LIN {X 0,Y 254.728,Z 728.451,A -85,B 0,C 180,E1 29641.69,E2 29641.69} C_VEL
LIN {X 0,Y 225.96,Z 695.224,A -85,B 0,C 180,E1 29666.244,E2 29666.244} C_VEL
LIN {X 0,Y 232.999,Z 658.239,A -85,B 0,C 180,E1 29686.941,E2 29686.941} C_VEL
LIN {X 0,Y 236.204,Z 647.926,A -85,B 0,C 180,E1 29697.112,E2 29697.112} C_VEL
LIN {X 0,Y 235.985,Z 649.701,A -85,B 0,C 180,E1 29705.085,E2 29705.085} C_VEL
LIN {X 0,Y 233.22,Z 662.932,A -85,B 0,C 180,E1 29715.199,E2 29715.199} C_VEL
LIN {X 0,Y 229.881,Z 671.076,A -85,B 0,C 180,E1 29718.505,E2 29718.505} C_VEL
LIN {X 0,Y 187.85,Z 714.712,A -85,B 0,C 180,E1 29726.634,E2 29726.634} C_VEL
LIN {X 0,Y 147.086,Z 745.833,A -85,B 0,C 180,E1 29741.377,E2 29741.377} C_VEL
LIN {X 0,Y 119.441,Z 763.935,A -85,B 0,C 180,E1 29767.61,E2 29767.61} C_VEL
LIN {X 0,Y 115.488,Z 767.444,A -85,B 0,C 180,E1 29793.764,E2 29793.764} C_VEL
LIN {X 0,Y 126.212,Z 759.493,A -85,B 0,C 180,E1 29822.73,E2 29822.73} C_VEL
LIN {X 0,Y 159.049,Z 737.597,A -85,B 0,C 180,E1 29844.139,E2 29844.139} C_VEL
LIN {X 0,Y 202.331,Z 701.352,A -85,B 0,C 180,E1 29856.657,E2 29856.657} C_VEL
LIN {X 0,Y 232.022,Z 667.67,A -85,B 0,C 180,E1 29862.272,E2 29862.272} C_VEL
LIN {X 0,Y 235.351,Z 652.826,A -85,B 0,C 180,E1 29871.562,E2 29871.562} C_VEL
LIN {X 0,Y 236.575,Z 647.685,A -85,B 0,C 180,E1 29878.052,E2 29878.052} C_VEL
LIN {X 0,Y 235.139,Z 650.478,A -85,B 0,C 180,E1 29886.517,E2 29886.517} C_VEL
LIN {X 0,Y 230.962,Z 664.925,A -85,B 0,C 180,E1 29897.076,E2 29897.076} C_VEL
LIN {X 0,Y 228.751,Z 702.6,A -85,B 0,C 180,E1 29918.911,E2 29918.911} C_VEL
LIN {X 0,Y 256.269,Z 729.185,A -85,B 0,C 180,E1 29938.946,E2 29938.946} C_VEL
LIN {X 0,Y 277.902,Z 744.199,A -85,B 0,C 180,E1 29950.33,E2 29950.33} C_VEL
LIN {X 0,Y 291.233,Z 754.024,A -85,B 0,C 180,E1 29959.499,E2 29959.499} C_VEL
LIN {X 0,Y 297.321,Z 758.46,A -85,B 0,C 180,E1 29968.539,E2 29968.539} C_VEL
LIN {X 0,Y 293.962,Z 756.258,A -85,B 0,C 180,E1 29977.41,E2 29977.41} C_VEL
LIN {X 0,Y 285.173,Z 749.557,A -85,B 0,C 180,E1 29985.141,E2 29985.141} C_VEL
LIN {X 0,Y 267.259,Z 737.135,A -85,B 0,C 180,E1 29995.187,E2 29995.187} C_VEL
LIN {X 0,Y 254.728,Z 728.451,A -85,B 0,C 180,E1 30001.69,E2 30001.69} C_VEL
LIN {X 0,Y 235.39,Z 722.248,A -85,B 0,C 180,E1 30008.545,E2 30008.545} C_VEL
LIN {X 0,Y 219.271,Z 687.766,A -85,B 0,C 180,E1 30034.122,E2 30034.122} C_VEL
LIN {X 0,Y 227.812,Z 663.177,A -85,B 0,C 180,E1 30047.874,E2 30047.874} C_VEL
LIN {X 0,Y 231.564,Z 653.613,A -85,B 0,C 180,E1 30058.235,E2 30058.235} C_VEL
LIN {X 0,Y 230.318,Z 658.459,A -85,B 0,C 180,E1 30067.685,E2 30067.685} C_VEL
LIN {X 0,Y 226.212,Z 672.442,A -85,B 0,C 180,E1 30076.746,E2 30076.746} C_VEL
LIN {X 0,Y 182.571,Z 716.057,A -85,B 0,C 180,E1 30084.791,E2 30084.791} C_VEL
LIN {X 0,Y 139.135,Z 747.341,A -85,B 0,C 180,E1 30100.274,E2 30100.274} C_VEL
LIN {X 0,Y 111.968,Z 763.757,A -85,B 0,C 180,E1 30126.026,E2 30126.026} C_VEL
LIN {X 0,Y 107.486,Z 767.269,A -85,B 0,C 180,E1 30154.045,E2 30154.045} C_VEL
LIN {X 0,Y 119.424,Z 759.314,A -85,B 0,C 180,E1 30184.849,E2 30184.849} C_VEL
LIN {X 0,Y 156.677,Z 735.903,A -85,B 0,C 180,E1 30207.488,E2 30207.488} C_VEL
LIN {X 0,Y 202.506,Z 698.173,A -85,B 0,C 180,E1 30219.402,E2 30219.402} C_VEL
LIN {X 0,Y 226.779,Z 671.402,A -85,B 0,C 180,E1 30223.58,E2 30223.58} C_VEL
LIN {X 0,Y 230.339,Z 658.433,A -85,B 0,C 180,E1 30232.316,E2 30232.316} C_VEL
LIN {X 0,Y 231.466,Z 653.736,A -85,B 0,C 180,E1 30241.766,E2 30241.766} C_VEL
LIN {X 0,Y 227.823,Z 663.166,A -85,B 0,C 180,E1 30252.127,E2 30252.127} C_VEL
LIN {X 0,Y 221.662,Z 706.254,A -85,B 0,C 180,E1 30278.627,E2 30278.627} C_VEL
LIN {X 0,Y 249.251,Z 732.077,A -85,B 0,C 180,E1 30299.507,E2 30299.507} C_VEL
LIN {X 0,Y 270.249,Z 745.742,A -85,B 0,C 180,E1 30310.718,E2 30310.718} C_VEL
LIN {X 0,Y 284.074,Z 755.281,A -85,B 0,C 180,E1 30320.563,E2 30320.563} C_VEL
LIN {X 0,Y 289.26,Z 758.636,A -85,B 0,C 180,E1 30328.498,E2 30328.498} C_VEL
LIN {X 0,Y 287.734,Z 757.916,A -85,B 0,C 180,E1 30334.534,E2 30334.534} C_VEL
LIN {X 0,Y 281.099,Z 753.131,A -85,B 0,C 180,E1 30342.16,E2 30342.16} C_VEL
LIN {X 0,Y 265.437,Z 742.878,A -85,B 0,C 180,E1 30351.799,E2 30351.799} C_VEL
LIN {X 0,Y 239.784,Z 725.609,A -85,B 0,C 180,E1 30365.759,E2 30365.759} C_VEL
LIN {X 0,Y 235.39,Z 722.248,A -85,B 0,C 180,E1 30368.545,E2 30368.545} C_VEL
LIN {X 0,Y 218.325,Z 716.283,A -85,B 0,C 180,E1 30376.29,E2 30376.29} C_VEL
LIN {X 0,Y 216.594,Z 681.525,A -85,B 0,C 180,E1 30400.946,E2 30400.946} C_VEL
LIN {X 0,Y 223.467,Z 666.107,A -85,B 0,C 180,E1 30410.346,E2 30410.346} C_VEL
LIN {X 0,Y 226.478,Z 659.971,A -85,B 0,C 180,E1 30418.196,E2 30418.196} C_VEL
LIN {X 0,Y 225.418,Z 663.045,A -85,B 0,C 180,E1 30425.911,E2 30425.911} C_VEL
LIN {X 0,Y 221.713,Z 674.444,A -85,B 0,C 180,E1 30434.56,E2 30434.56} C_VEL
LIN {X 0,Y 178.102,Z 716.889,A -85,B 0,C 180,E1 30442.7,E2 30442.7} C_VEL
LIN {X 0,Y 134.023,Z 747.163,A -85,B 0,C 180,E1 30457.621,E2 30457.621} C_VEL
LIN {X 0,Y 104.613,Z 763.58,A -85,B 0,C 180,E1 30484.222,E2 30484.222} C_VEL
LIN {X 0,Y 99.454,Z 767.059,A -85,B 0,C 180,E1 30515.015,E2 30515.015} C_VEL
LIN {X 0,Y 114.521,Z 758.116,A -85,B 0,C 180,E1 30548.976,E2 30548.976} C_VEL
LIN {X 0,Y 153.452,Z 735.034,A -85,B 0,C 180,E1 30570.429,E2 30570.429} C_VEL
LIN {X 0,Y 199.79,Z 697.995,A -85,B 0,C 180,E1 30581.586,E2 30581.586} C_VEL
LIN {X 0,Y 221.953,Z 674.175,A -85,B 0,C 180,E1 30585.469,E2 30585.469} C_VEL
LIN {X 0,Y 225.412,Z 663.051,A -85,B 0,C 180,E1 30594.089,E2 30594.089} C_VEL
LIN {X 0,Y 226.375,Z 660.091,A -85,B 0,C 180,E1 30601.805,E2 30601.805} C_VEL
LIN {X 0,Y 221.763,Z 670.312,A -85,B 0,C 180,E1 30612.726,E2 30612.726} C_VEL
LIN {X 0,Y 214.375,Z 709.528,A -85,B 0,C 180,E1 30638.119,E2 30638.119} C_VEL
LIN {X 0,Y 242.903,Z 735.294,A -85,B 0,C 180,E1 30660.516,E2 30660.516} C_VEL
LIN {X 0,Y 263.361,Z 747.739,A -85,B 0,C 180,E1 30671.592,E2 30671.592} C_VEL
LIN {X 0,Y 275.604,Z 755.471,A -85,B 0,C 180,E1 30680.271,E2 30680.271} C_VEL
LIN {X 0,Y 281.172,Z 758.813,A -85,B 0,C 180,E1 30688.455,E2 30688.455} C_VEL
LIN {X 0,Y 279.558,Z 758.096,A -85,B 0,C 180,E1 30694.667,E2 30694.667} C_VEL
LIN {X 0,Y 271.859,Z 753.075,A -85,B 0,C 180,E1 30702.843,E2 30702.843} C_VEL
LIN {X 0,Y 254.88,Z 742.852,A -85,B 0,C 180,E1 30712.945,E2 30712.945} C_VEL
LIN {X 0,Y 227.506,Z 724.851,A -85,B 0,C 180,E1 30728.684,E2 30728.684} C_VEL
LIN {X 0,Y 218.325,Z 716.283,A -85,B 0,C 180,E1 30736.29,E2 30736.29} C_VEL
LIN {X 0,Y 205.918,Z 709.678,A -85,B 0,C 180,E1 30745.1,E2 30745.1} C_VEL
LIN {X 0,Y 217.606,Z 672.647,A -85,B 0,C 180,E1 30770.083,E2 30770.083} C_VEL
LIN {X 0,Y 221.058,Z 666.041,A -85,B 0,C 180,E1 30778.151,E2 30778.151} C_VEL
LIN {X 0,Y 219.856,Z 669.284,A -85,B 0,C 180,E1 30786.061,E2 30786.061} C_VEL
LIN {X 0,Y 216.387,Z 678.218,A -85,B 0,C 180,E1 30793.213,E2 30793.213} C_VEL
LIN {X 0,Y 170.784,Z 720.013,A -85,B 0,C 180,E1 30801.194,E2 30801.194} C_VEL
LIN {X 0,Y 124.008,Z 749.858,A -85,B 0,C 180,E1 30817.356,E2 30817.356} C_VEL
LIN {X 0,Y 95.225,Z 764.536,A -85,B 0,C 180,E1 30846.538,E2 30846.538} C_VEL
LIN {X 0,Y 91.484,Z 766.918,A -85,B 0,C 180,E1 30874.754,E2 30874.754} C_VEL
LIN {X 0,Y 106.426,Z 758.957,A -85,B 0,C 180,E1 30909.882,E2 30909.882} C_VEL
LIN {X 0,Y 148.984,Z 735.263,A -85,B 0,C 180,E1 30932.955,E2 30932.955} C_VEL
LIN {X 0,Y 197.378,Z 697.818,A -85,B 0,C 180,E1 30943.821,E2 30943.821} C_VEL
LIN {X 0,Y 216.834,Z 677.517,A -85,B 0,C 180,E1 30947.079,E2 30947.079} C_VEL
LIN {X 0,Y 220.44,Z 667.708,A -85,B 0,C 180,E1 30955.951,E2 30955.951} C_VEL
LIN {X 0,Y 220.308,Z 667.079,A -85,B 0,C 180,E1 30963.529,E2 30963.529} C_VEL
LIN {X 0,Y 215.403,Z 676.961,A -85,B 0,C 180,E1 30973.109,E2 30973.109} C_VEL
LIN {X 0,Y 207.451,Z 713.563,A -85,B 0,C 180,E1 30998.277,E2 30998.277} C_VEL
LIN {X 0,Y 235.856,Z 737.914,A -85,B 0,C 180,E1 31021.169,E2 31021.169} C_VEL
LIN {X 0,Y 256.839,Z 749.754,A -85,B 0,C 180,E1 31032.751,E2 31032.751} C_VEL
LIN {X 0,Y 268.905,Z 756.817,A -85,B 0,C 180,E1 31041.895,E2 31041.895} C_VEL
LIN {X 0,Y 273.109,Z 758.99,A -85,B 0,C 180,E1 31048.409,E2 31048.409} C_VEL
LIN {X 0,Y 271.34,Z 758.278,A -85,B 0,C 180,E1 31054.809,E2 31054.809} C_VEL
LIN {X 0,Y 262.883,Z 753.278,A -85,B 0,C 180,E1 31063.289,E2 31063.289} C_VEL
LIN {X 0,Y 245.026,Z 743.359,A -85,B 0,C 180,E1 31073.722,E2 31073.722} C_VEL
LIN {X 0,Y 217.8,Z 726.02,A -85,B 0,C 180,E1 31090.169,E2 31090.169} C_VEL
LIN {X 0,Y 205.918,Z 709.678,A -85,B 0,C 180,E1 31105.1,E2 31105.1} C_VEL
LIN {X 0,Y 199.485,Z 701.993,A -85,B 0,C 180,E1 31114.737,E2 31114.737} C_VEL
LIN {X 0,Y 212.093,Z 677.669,A -85,B 0,C 180,E1 31130.862,E2 31130.862} C_VEL
LIN {X 0,Y 215.64,Z 672.089,A -85,B 0,C 180,E1 31138.105,E2 31138.105} C_VEL
LIN {X 0,Y 214.136,Z 675.443,A -85,B 0,C 180,E1 31146.223,E2 31146.223} C_VEL
LIN {X 0,Y 210.393,Z 682.827,A -85,B 0,C 180,E1 31151.881,E2 31151.881} C_VEL
LIN {X 0,Y 163.045,Z 723.354,A -85,B 0,C 180,E1 31159.655,E2 31159.655} C_VEL
LIN {X 0,Y 116.019,Z 751.214,A -85,B 0,C 180,E1 31175.896,E2 31175.896} C_VEL
LIN {X 0,Y 87.861,Z 764.36,A -85,B 0,C 180,E1 31204.437,E2 31204.437} C_VEL
LIN {X 0,Y 83.47,Z 766.742,A -85,B 0,C 180,E1 31235.211,E2 31235.211} C_VEL
LIN {X 0,Y 100.289,Z 758.779,A -85,B 0,C 180,E1 31272.879,E2 31272.879} C_VEL
LIN {X 0,Y 145.43,Z 735.084,A -85,B 0,C 180,E1 31295.841,E2 31295.841} C_VEL
LIN {X 0,Y 195.273,Z 697.641,A -85,B 0,C 180,E1 31306.106,E2 31306.106} C_VEL
LIN {X 0,Y 211.826,Z 680.845,A -85,B 0,C 180,E1 31308.851,E2 31308.851} C_VEL
LIN {X 0,Y 215.556,Z 672.545,A -85,B 0,C 180,E1 31317.862,E2 31317.862} C_VEL
LIN {X 0,Y 213.738,Z 674.762,A -85,B 0,C 180,E1 31325.99,E2 31325.99} C_VEL
LIN {X 0,Y 206.613,Z 687.133,A -85,B 0,C 180,E1 31335.63,E2 31335.63} C_VEL
LIN {X 0,Y 201.148,Z 718.649,A -85,B 0,C 180,E1 31359.708,E2 31359.708} C_VEL
LIN {X 0,Y 230.107,Z 741.108,A -85,B 0,C 180,E1 31382.642,E2 31382.642} C_VEL
LIN {X 0,Y 250.759,Z 751.859,A -85,B 0,C 180,E1 31394.208,E2 31394.208} C_VEL
LIN {X 0,Y 260.559,Z 757.003,A -85,B 0,C 180,E1 31401.634,E2 31401.634} C_VEL
LIN {X 0,Y 265.004,Z 759.167,A -85,B 0,C 180,E1 31408.361,E2 31408.361} C_VEL
LIN {X 0,Y 263.113,Z 758.46,A -85,B 0,C 180,E1 31414.96,E2 31414.96} C_VEL
LIN {X 0,Y 253.467,Z 753.325,A -85,B 0,C 180,E1 31423.971,E2 31423.971} C_VEL
LIN {X 0,Y 234.404,Z 743.612,A -85,B 0,C 180,E1 31434.868,E2 31434.868} C_VEL
LIN {X 0,Y 205.25,Z 724.518,A -85,B 0,C 180,E1 31454.581,E2 31454.581} C_VEL
LIN {X 0,Y 199.485,Z 701.993,A -85,B 0,C 180,E1 31474.737,E2 31474.737} C_VEL
LIN {X 0,Y 199.798,Z 692.818,A -85,B 0,C 180,E1 31484.582,E2 31484.582} C_VEL
LIN {X 0,Y 207.901,Z 680.595,A -85,B 0,C 180,E1 31493.841,E2 31493.841} C_VEL
LIN {X 0,Y 209.887,Z 677.873,A -85,B 0,C 180,E1 31498.053,E2 31498.053} C_VEL
LIN {X 0,Y 208.209,Z 681.369,A -85,B 0,C 180,E1 31506.401,E2 31506.401} C_VEL
LIN {X 0,Y 204.322,Z 687.264,A -85,B 0,C 180,E1 31510.23,E2 31510.23} C_VEL
LIN {X 0,Y 155.19,Z 726.857,A -85,B 0,C 180,E1 31518.046,E2 31518.046} C_VEL
LIN {X 0,Y 106.489,Z 753.364,A -85,B 0,C 180,E1 31535.189,E2 31535.189} C_VEL
LIN {X 0,Y 76.779,Z 765.765,A -85,B 0,C 180,E1 31572.766,E2 31572.766} C_VEL
LIN {X 0,Y 76.798,Z 765.765,A -85,B 0,C 180,E1 31607.229,E2 31607.229} C_VEL
LIN {X 0,Y 106.401,Z 753.393,A -85,B 0,C 180,E1 31644.793,E2 31644.793} C_VEL
LIN {X 0,Y 156.662,Z 725.837,A -85,B 0,C 180,E1 31662.297,E2 31662.297} C_VEL
LIN {X 0,Y 206.169,Z 685.486,A -85,B 0,C 180,E1 31670,E2 31670} C_VEL
LIN {X 0,Y 209.786,Z 678.334,A -85,B 0,C 180,E1 31677.803,E2 31677.803} C_VEL
LIN {X 0,Y 208.766,Z 679.221,A -85,B 0,C 180,E1 31684.043,E2 31684.043} C_VEL
LIN {X 0,Y 202.748,Z 688.544,A -85,B 0,C 180,E1 31692.9,E2 31692.9} C_VEL
LIN {X 0,Y 193.386,Z 721.096,A -85,B 0,C 180,E1 31718.661,E2 31718.661} C_VEL
LIN {X 0,Y 220.27,Z 741.933,A -85,B 0,C 180,E1 31741.778,E2 31741.778} C_VEL
LIN {X 0,Y 243.246,Z 752.979,A -85,B 0,C 180,E1 31754.78,E2 31754.78} C_VEL
LIN {X 0,Y 252.476,Z 757.404,A -85,B 0,C 180,E1 31761.786,E2 31761.786} C_VEL
LIN {X 0,Y 256.875,Z 759.345,A -85,B 0,C 180,E1 31768.309,E2 31768.309} C_VEL
LIN {X 0,Y 254.845,Z 758.642,A -85,B 0,C 180,E1 31775.121,E2 31775.121} C_VEL
LIN {X 0,Y 245.339,Z 754.088,A -85,B 0,C 180,E1 31783.771,E2 31783.771} C_VEL
LIN {X 0,Y 225.561,Z 744.821,A -85,B 0,C 180,E1 31795.035,E2 31795.035} C_VEL
LIN {X 0,Y 196.549,Z 726.274,A -85,B 0,C 180,E1 31815.926,E2 31815.926} C_VEL
LIN {X 0,Y 198.212,Z 695.345,A -85,B 0,C 180,E1 31843.011,E2 31843.011} C_VEL
LIN {X 0,Y 199.798,Z 692.818,A -85,B 0,C 180,E1 31844.582,E2 31844.582} C_VEL
LIN {X 0,Y 202.236,Z 685.819,A -85,B 0,C 180,E1 31854.611,E2 31854.611} C_VEL
LIN {X 0,Y 204.067,Z 683.66,A -85,B 0,C 180,E1 31857.997,E2 31857.997} C_VEL
LIN {X 0,Y 203.221,Z 685.374,A -85,B 0,C 180,E1 31864.215,E2 31864.215} C_VEL
LIN {X 0,Y 199.657,Z 690.226,A -85,B 0,C 180,E1 31868.341,E2 31868.341} C_VEL
LIN {X 0,Y 147.973,Z 729.601,A -85,B 0,C 180,E1 31876.098,E2 31876.098} C_VEL
LIN {X 0,Y 96.642,Z 755.344,A -85,B 0,C 180,E1 31894.53,E2 31894.53} C_VEL
LIN {X 0,Y 69.101,Z 765.588,A -85,B 0,C 180,E1 31930.78,E2 31930.78} C_VEL
LIN {X 0,Y 69.137,Z 765.589,A -85,B 0,C 180,E1 31969.209,E2 31969.209} C_VEL
LIN {X 0,Y 102.069,Z 753.138,A -85,B 0,C 180,E1 32008.647,E2 32008.647} C_VEL
LIN {X 0,Y 154.28,Z 725.724,A -85,B 0,C 180,E1 32025.167,E2 32025.167} C_VEL
LIN {X 0,Y 201.651,Z 688.062,A -85,B 0,C 180,E1 32032.501,E2 32032.501} C_VEL
LIN {X 0,Y 203.979,Z 684.108,A -85,B 0,C 180,E1 32037.741,E2 32037.741} C_VEL
LIN {X 0,Y 203.077,Z 684.785,A -85,B 0,C 180,E1 32043.757,E2 32043.757} C_VEL
LIN {X 0,Y 196.291,Z 693.939,A -85,B 0,C 180,E1 32052.561,E2 32052.561} C_VEL
LIN {X 0,Y 186.512,Z 725.125,A -85,B 0,C 180,E1 32079.428,E2 32079.428} C_VEL
LIN {X 0,Y 216.109,Z 745.558,A -85,B 0,C 180,E1 32104.259,E2 32104.259} C_VEL
LIN {X 0,Y 234.036,Z 753.325,A -85,B 0,C 180,E1 32114.324,E2 32114.324} C_VEL
LIN {X 0,Y 243.304,Z 757.389,A -85,B 0,C 180,E1 32121.036,E2 32121.036} C_VEL
LIN {X 0,Y 248.744,Z 759.522,A -85,B 0,C 180,E1 32128.253,E2 32128.253} C_VEL
LIN {X 0,Y 246.557,Z 758.825,A -85,B 0,C 180,E1 32135.294,E2 32135.294} C_VEL
LIN {X 0,Y 238.261,Z 755.22,A -85,B 0,C 180,E1 32142.872,E2 32142.872} C_VEL
LIN {X 0,Y 218.727,Z 746.935,A -85,B 0,C 180,E1 32154.094,E2 32154.094} C_VEL
LIN {X 0,Y 189.194,Z 729.369,A -85,B 0,C 180,E1 32175.802,E2 32175.802} C_VEL
LIN {X 0,Y 192.268,Z 699.14,A -85,B 0,C 180,E1 32204.108,E2 32204.108} C_VEL
LIN {X 0,Y 201.715,Z 686.519,A -85,B 0,C 180,E1 32213.652,E2 32213.652} C_VEL
LIN {X 0,Y 202.236,Z 685.819,A -85,B 0,C 180,E1 32214.611,E2 32214.611} C_VEL
LIN {X 0,Y 199.741,Z 687.736,A -85,B 0,C 180,E1 32220.845,E2 32220.845} C_VEL
LIN {X 0,Y 196.779,Z 691.204,A -85,B 0,C 180,E1 32224.687,E2 32224.687} C_VEL
LIN {X 0,Y 192.694,Z 695.503,A -85,B 0,C 180,E1 32226.61,E2 32226.61} C_VEL
LIN {X 0,Y 140.689,Z 732.503,A -85,B 0,C 180,E1 32234.042,E2 32234.042} C_VEL
LIN {X 0,Y 89.421,Z 756.194,A -85,B 0,C 180,E1 32252.01,E2 32252.01} C_VEL
LIN {X 0,Y 61.525,Z 765.411,A -85,B 0,C 180,E1 32288.301,E2 32288.301} C_VEL
LIN {X 0,Y 61.555,Z 765.412,A -85,B 0,C 180,E1 32331.687,E2 32331.687} C_VEL
LIN {X 0,Y 98.096,Z 752.949,A -85,B 0,C 180,E1 32372.735,E2 32372.735} C_VEL
LIN {X 0,Y 151.716,Z 725.995,A -85,B 0,C 180,E1 32388.019,E2 32388.019} C_VEL
LIN {X 0,Y 196.221,Z 692.141,A -85,B 0,C 180,E1 32394.061,E2 32394.061} C_VEL
LIN {X 0,Y 197.827,Z 689.304,A -85,B 0,C 180,E1 32402.066,E2 32402.066} C_VEL
LIN {X 0,Y 190.666,Z 697.871,A -85,B 0,C 180,E1 32411.335,E2 32411.335} C_VEL
LIN {X 0,Y 179.083,Z 728.149,A -85,B 0,C 180,E1 32439.262,E2 32439.262} C_VEL
LIN {X 0,Y 208.813,Z 747.467,A -85,B 0,C 180,E1 32464.966,E2 32464.966} C_VEL
LIN {X 0,Y 228.932,Z 755.432,A -85,B 0,C 180,E1 32476.594,E2 32476.594} C_VEL
LIN {X 0,Y 238.105,Z 759.012,A -85,B 0,C 180,E1 32484.518,E2 32484.518} C_VEL
LIN {X 0,Y 240.556,Z 759.702,A -85,B 0,C 180,E1 32491.806,E2 32491.806} C_VEL
LIN {X 0,Y 232.853,Z 756.938,A -85,B 0,C 180,E1 32500.695,E2 32500.695} C_VEL
LIN {X 0,Y 214.366,Z 749.866,A -85,B 0,C 180,E1 32511.754,E2 32511.754} C_VEL
LIN {X 0,Y 184.349,Z 734.606,A -85,B 0,C 180,E1 32532.559,E2 32532.559} C_VEL
LIN {X 0,Y 184.485,Z 705.482,A -85,B 0,C 180,E1 32563.419,E2 32563.419} C_VEL
LIN {X 0,Y 195.211,Z 692.31,A -85,B 0,C 180,E1 32573.439,E2 32573.439} C_VEL
LIN {X 0,Y 197.972,Z 689.176,A -85,B 0,C 180,E1 32577.936,E2 32577.936} C_VEL
LIN {X 0,Y 196.779,Z 691.204,A -85,B 0,C 180,E1 32584.687,E2 32584.687} C_VEL
LIN {X 0,Y 189.449,Z 697.862,A -85,B 0,C 180,E1 32585.726,E2 32585.726} C_VEL
LIN {X 0,Y 178.401,Z 706.412,A -85,B 0,C 180,E1 32585.494,E2 32585.494} C_VEL
LIN {X 0,Y 124.402,Z 739.949,A -85,B 0,C 180,E1 32593.744,E2 32593.744} C_VEL
LIN {X 0,Y 74.046,Z 759.677,A -85,B 0,C 180,E1 32614.993,E2 32614.993} C_VEL
LIN {X 0,Y 51.354,Z 766.036,A -85,B 0,C 180,E1 32661.508,E2 32661.508} C_VEL
LIN {X 0,Y 64.306,Z 762.508,A -85,B 0,C 180,E1 32715.079,E2 32715.079} C_VEL
LIN {X 0,Y 114.509,Z 744.576,A -85,B 0,C 180,E1 32743.768,E2 32743.768} C_VEL
LIN {X 0,Y 169.769,Z 712.734,A -85,B 0,C 180,E1 32753.594,E2 32753.594} C_VEL
LIN {X 0,Y 190.108,Z 696.931,A -85,B 0,C 180,E1 32755.649,E2 32755.649} C_VEL
LIN {X 0,Y 191.615,Z 694.804,A -85,B 0,C 180,E1 32762.133,E2 32762.133} C_VEL
LIN {X 0,Y 183.803,Z 703.06,A -85,B 0,C 180,E1 32771.024,E2 32771.024} C_VEL
LIN {X 0,Y 171.752,Z 731.326,A -85,B 0,C 180,E1 32799.352,E2 32799.352} C_VEL
LIN {X 0,Y 201.111,Z 749.136,A -85,B 0,C 180,E1 32825.498,E2 32825.498} C_VEL
LIN {X 0,Y 219.601,Z 755.644,A -85,B 0,C 180,E1 32836.013,E2 32836.013} C_VEL
LIN {X 0,Y 229.721,Z 759.198,A -85,B 0,C 180,E1 32844.317,E2 32844.317} C_VEL
LIN {X 0,Y 232.372,Z 759.881,A -85,B 0,C 180,E1 32851.87,E2 32851.87} C_VEL
LIN {X 0,Y 223.718,Z 757.164,A -85,B 0,C 180,E1 32861.089,E2 32861.089} C_VEL
LIN {X 0,Y 204.565,Z 750.536,A -85,B 0,C 180,E1 32872.351,E2 32872.351} C_VEL
LIN {X 0,Y 173.957,Z 734.75,A -85,B 0,C 180,E1 32895.966,E2 32895.966} C_VEL
LIN {X 0,Y 180.883,Z 706.241,A -85,B 0,C 180,E1 32926.825,E2 32926.825} C_VEL
LIN {X 0,Y 190.185,Z 696.278,A -85,B 0,C 180,E1 32935.36,E2 32935.36} C_VEL
LIN {X 0,Y 191.692,Z 695.097,A -85,B 0,C 180,E1 32942.404,E2 32942.404} C_VEL
LIN {X 0,Y 188.731,Z 698.051,A -85,B 0,C 180,E1 32944.498,E2 32944.498} C_VEL
LIN {X 0,Y 178.401,Z 706.412,A -85,B 0,C 180,E1 32945.494,E2 32945.494} C_VEL
LIN {X 0,Y 148.742,Z 725.885,A -85,B 0,C 180,E1 32945.933,E2 32945.933} C_VEL
LIN {X 0,Y 91.802,Z 752.594,A -85,B 0,C 180,E1 32958.221,E2 32958.221} C_VEL
LIN {X 0,Y 46.888,Z 765.058,A -85,B 0,C 180,E1 33000.977,E2 33000.977} C_VEL
LIN {X 0,Y 43.565,Z 765.863,A -85,B 0,C 180,E1 33040.022,E2 33040.022} C_VEL
LIN {X 0,Y 75.652,Z 757.886,A -85,B 0,C 180,E1 33094.428,E2 33094.428} C_VEL
LIN {X 0,Y 134.004,Z 734.192,A -85,B 0,C 180,E1 33111.976,E2 33111.976} C_VEL
LIN {X 0,Y 185.409,Z 700.088,A -85,B 0,C 180,E1 33118.165,E2 33118.165} C_VEL
LIN {X 0,Y 183.373,Z 701.639,A -85,B 0,C 180,E1 33124.642,E2 33124.642} C_VEL
LIN {X 0,Y 164.671,Z 734.777,A -85,B 0,C 180,E1 33160.254,E2 33160.254} C_VEL
LIN {X 0,Y 191.794,Z 750.093,A -85,B 0,C 180,E1 33185.142,E2 33185.142} C_VEL
LIN {X 0,Y 210.67,Z 756.171,A -85,B 0,C 180,E1 33195.952,E2 33195.952} C_VEL
LIN {X 0,Y 221.161,Z 759.387,A -85,B 0,C 180,E1 33204.097,E2 33204.097} C_VEL
LIN {X 0,Y 224.192,Z 760.059,A -85,B 0,C 180,E1 33208.062,E2 33208.062} C_VEL
LIN {X 0,Y 221.233,Z 759.385,A -85,B 0,C 180,E1 33215.902,E2 33215.902} C_VEL
LIN {X 0,Y 209.356,Z 755.878,A -85,B 0,C 180,E1 33224.686,E2 33224.686} C_VEL
LIN {X 0,Y 183.378,Z 747.07,A -85,B 0,C 180,E1 33239.973,E2 33239.973} C_VEL
LIN {X 0,Y 164.632,Z 722.855,A -85,B 0,C 180,E1 33275.673,E2 33275.673} C_VEL
LIN {X 0,Y 183.343,Z 701.686,A -85,B 0,C 180,E1 33295.187,E2 33295.187} C_VEL
LIN {X 0,Y 185.414,Z 700.057,A -85,B 0,C 180,E1 33301.654,E2 33301.654} C_VEL
LIN {X 0,Y 148.742,Z 725.885,A -85,B 0,C 180,E1 33305.933,E2 33305.933} C_VEL
LIN {X 0,Y 117.077,Z 741.688,A -85,B 0,C 180,E1 33307,E2 33307} C_VEL
LIN {X 0,Y 59.86,Z 760.913,A -85,B 0,C 180,E1 33327.539,E2 33327.539} C_VEL
LIN {X 0,Y 35.511,Z 765.684,A -85,B 0,C 180,E1 33377.67,E2 33377.67} C_VEL
LIN {X 0,Y 54.025,Z 762.158,A -85,B 0,C 180,E1 33447.362,E2 33447.362} C_VEL
LIN {X 0,Y 110.58,Z 744.422,A -85,B 0,C 180,E1 33471.769,E2 33471.769} C_VEL
LIN {X 0,Y 168.73,Z 712.378,A -85,B 0,C 180,E1 33479.096,E2 33479.096} C_VEL
LIN {X 0,Y 178.953,Z 704.942,A -85,B 0,C 180,E1 33480.308,E2 33480.308} C_VEL
LIN {X 0,Y 172.555,Z 710.349,A -85,B 0,C 180,E1 33488.221,E2 33488.221} C_VEL
LIN {X 0,Y 156.632,Z 736.634,A -85,B 0,C 180,E1 33518.809,E2 33518.809} C_VEL
LIN {X 0,Y 187.745,Z 752.829,A -85,B 0,C 180,E1 33547.96,E2 33547.96} C_VEL
LIN {X 0,Y 207.682,Z 758.303,A -85,B 0,C 180,E1 33559.753,E2 33559.753} C_VEL
LIN {X 0,Y 215.919,Z 760.24,A -85,B 0,C 180,E1 33567.988,E2 33567.988} C_VEL
LIN {X 0,Y 215.903,Z 760.241,A -85,B 0,C 180,E1 33572.013,E2 33572.013} C_VEL
LIN {X 0,Y 207.161,Z 758.199,A -85,B 0,C 180,E1 33580.545,E2 33580.545} C_VEL
LIN {X 0,Y 187.604,Z 752.925,A -85,B 0,C 180,E1 33591.934,E2 33591.934} C_VEL
LIN {X 0,Y 155.715,Z 735.029,A -85,B 0,C 180,E1 33623.894,E2 33623.894} C_VEL
LIN {X 0,Y 176.85,Z 706.721,A -85,B 0,C 180,E1 33655.427,E2 33655.427} C_VEL
LIN {X 0,Y 178.981,Z 704.92,A -85,B 0,C 180,E1 33659.705,E2 33659.705} C_VEL
LIN {X 0,Y 122.023,Z 739.366,A -85,B 0,C 180,E1 33666.153,E2 33666.153} C_VEL
LIN {X 0,Y 117.077,Z 741.688,A -85,B 0,C 180,E1 33667,E2 33667} C_VEL
LIN {X 0,Y 83.788,Z 753.608,A -85,B 0,C 180,E1 33669.138,E2 33669.138} C_VEL
LIN {X 0,Y 33.685,Z 764.705,A -85,B 0,C 180,E1 33707.522,E2 33707.522} C_VEL
LIN {X 0,Y 27.834,Z 765.511,A -85,B 0,C 180,E1 33765.807,E2 33765.807} C_VEL
LIN {X 0,Y 70.172,Z 757.53,A -85,B 0,C 180,E1 33826.529,E2 33826.529} C_VEL
LIN {X 0,Y 132.353,Z 734.018,A -85,B 0,C 180,E1 33838.925,E2 33838.925} C_VEL
LIN {X 0,Y 171.576,Z 710.274,A -85,B 0,C 180,E1 33842.382,E2 33842.382} C_VEL
LIN {X 0,Y 149.878,Z 740.457,A -85,B 0,C 180,E1 33880.917,E2 33880.917} C_VEL
LIN {X 0,Y 177.92,Z 753.555,A -85,B 0,C 180,E1 33907.446,E2 33907.446} C_VEL
LIN {X 0,Y 197.822,Z 758.409,A -85,B 0,C 180,E1 33918.951,E2 33918.951} C_VEL
LIN {X 0,Y 207.589,Z 760.422,A -85,B 0,C 180,E1 33927.907,E2 33927.907} C_VEL
LIN {X 0,Y 205.187,Z 760.058,A -85,B 0,C 180,E1 33935.118,E2 33935.118} C_VEL
LIN {X 0,Y 194.229,Z 757.686,A -85,B 0,C 180,E1 33943.07,E2 33943.07} C_VEL
LIN {X 0,Y 169.411,Z 751.084,A -85,B 0,C 180,E1 33957.769,E2 33957.769} C_VEL
LIN {X 0,Y 150.847,Z 728.866,A -85,B 0,C 180,E1 33997.707,E2 33997.707} C_VEL
LIN {X 0,Y 171.672,Z 710.207,A -85,B 0,C 180,E1 34017.619,E2 34017.619} C_VEL
LIN {X 0,Y 113.933,Z 742.522,A -85,B 0,C 180,E1 34023.356,E2 34023.356} C_VEL
LIN {X 0,Y 83.788,Z 753.608,A -85,B 0,C 180,E1 34029.138,E2 34029.138} C_VEL
LIN {X 0,Y 49.635,Z 761.379,A -85,B 0,C 180,E1 34034.419,E2 34034.419} C_VEL
LIN {X 0,Y 20.09,Z 765.332,A -85,B 0,C 180,E1 34087.824,E2 34087.824} C_VEL
LIN {X 0,Y 40.515,Z 762.94,A -85,B 0,C 180,E1 34179.346,E2 34179.346} C_VEL
LIN {X 0,Y 103.162,Z 746.58,A -85,B 0,C 180,E1 34199.512,E2 34199.512} C_VEL
LIN {X 0,Y 162.154,Z 716.909,A -85,B 0,C 180,E1 34204.596,E2 34204.596} C_VEL
LIN {X 0,Y 141.737,Z 742.179,A -85,B 0,C 180,E1 34239.521,E2 34239.521} C_VEL
LIN {X 0,Y 170.723,Z 754.943,A -85,B 0,C 180,E1 34268.508,E2 34268.508} C_VEL
LIN {X 0,Y 191.62,Z 759.422,A -85,B 0,C 180,E1 34280.878,E2 34280.878} C_VEL
LIN {X 0,Y 199.265,Z 760.604,A -85,B 0,C 180,E1 34287.819,E2 34287.819} C_VEL
LIN {X 0,Y 199.281,Z 760.604,A -85,B 0,C 180,E1 34292.181,E2 34292.181} C_VEL
LIN {X 0,Y 187.684,Z 758.638,A -85,B 0,C 180,E1 34301.654,E2 34301.654} C_VEL
LIN {X 0,Y 161.521,Z 752.596,A -85,B 0,C 180,E1 34317.183,E2 34317.183} C_VEL
LIN {X 0,Y 143.837,Z 732.034,A -85,B 0,C 180,E1 34358.529,E2 34358.529} C_VEL
LIN {X 0,Y 162.048,Z 716.969,A -85,B 0,C 180,E1 34375.477,E2 34375.477} C_VEL
LIN {X 0,Y 103.075,Z 746.614,A -85,B 0,C 180,E1 34380.485,E2 34380.485} C_VEL
LIN {X 0,Y 49.635,Z 761.379,A -85,B 0,C 180,E1 34394.419,E2 34394.419} C_VEL
LIN {X 0,Y 16.11,Z 764.885,A -85,B 0,C 180,E1 34417.974,E2 34417.974} C_VEL
LIN {X 0,Y 27.773,Z 764.004,A -85,B 0,C 180,E1 34543.171,E2 34543.171} C_VEL
LIN {X 0,Y 91.112,Z 750.613,A -85,B 0,C 180,E1 34562.982,E2 34562.982} C_VEL
LIN {X 0,Y 149.657,Z 724.891,A -85,B 0,C 180,E1 34567.43,E2 34567.43} C_VEL
LIN {X 0,Y 136.801,Z 747.176,A -85,B 0,C 180,E1 34605.854,E2 34605.854} C_VEL
LIN {X 0,Y 167.189,Z 757.006,A -85,B 0,C 180,E1 34631.831,E2 34631.831} C_VEL
LIN {X 0,Y 185.652,Z 760.174,A -85,B 0,C 180,E1 34642.962,E2 34642.962} C_VEL
LIN {X 0,Y 190.717,Z 760.791,A -85,B 0,C 180,E1 34647.722,E2 34647.722} C_VEL
LIN {X 0,Y 189.53,Z 760.721,A -85,B 0,C 180,E1 34653.398,E2 34653.398} C_VEL
LIN {X 0,Y 177.23,Z 758.874,A -85,B 0,C 180,E1 34662.352,E2 34662.352} C_VEL
LIN {X 0,Y 145.37,Z 751.526,A -85,B 0,C 180,E1 34683.187,E2 34683.187} C_VEL
LIN {X 0,Y 141.877,Z 730.342,A -85,B 0,C 180,E1 34726.158,E2 34726.158} C_VEL
LIN {X 0,Y 150.125,Z 724.541,A -85,B 0,C 180,E1 34733.046,E2 34733.046} C_VEL
LIN {X 0,Y 87.285,Z 751.882,A -85,B 0,C 180,E1 34737.447,E2 34737.447} C_VEL
LIN {X 0,Y 24.343,Z 764.351,A -85,B 0,C 180,E1 34760.854,E2 34760.854} C_VEL
LIN {X 0,Y 16.11,Z 764.885,A -85,B 0,C 180,E1 34777.974,E2 34777.974} C_VEL
LIN {X 0,Y 21.925,Z 764.219,A -85,B 0,C 180,E1 34918.211,E2 34918.211} C_VEL
LIN {X 0,Y 88.03,Z 751.705,A -85,B 0,C 180,E1 34927.889,E2 34927.889} C_VEL
LIN {X 0,Y 138.215,Z 731.427,A -85,B 0,C 180,E1 34929.933,E2 34929.933} C_VEL
LIN {X 0,Y 132.064,Z 750.899,A -85,B 0,C 180,E1 34970.835,E2 34970.835} C_VEL
LIN {X 0,Y 164.065,Z 758.76,A -85,B 0,C 180,E1 34995.519,E2 34995.519} C_VEL
LIN {X 0,Y 175.944,Z 760.389,A -85,B 0,C 180,E1 35002.572,E2 35002.572} C_VEL
LIN {X 0,Y 182.198,Z 760.978,A -85,B 0,C 180,E1 35007.615,E2 35007.615} C_VEL
LIN {X 0,Y 182.216,Z 760.978,A -85,B 0,C 180,E1 35012.385,E2 35012.385} C_VEL
LIN {X 0,Y 175.573,Z 760.361,A -85,B 0,C 180,E1 35017.614,E2 35017.614} C_VEL
LIN {X 0,Y 149.892,Z 756.239,A -85,B 0,C 180,E1 35032.942,E2 35032.942} C_VEL
LIN {X 0,Y 130.055,Z 737.375,A -85,B 0,C 180,E1 35081.105,E2 35081.105} C_VEL
LIN {X 0,Y 138.091,Z 731.483,A -85,B 0,C 180,E1 35090.124,E2 35090.124} C_VEL
LIN {X 0,Y 76.448,Z 754.948,A -85,B 0,C 180,E1 35092.683,E2 35092.683} C_VEL
LIN {X 0,Y 11.856,Z 764.762,A -85,B 0,C 180,E1 35109.616,E2 35109.616} C_VEL
LIN {X 0,Y 21.925,Z 764.219,A -85,B 0,C 180,E1 35278.211,E2 35278.211} C_VEL
LIN {X 0,Y 55.897,Z 759.774,A -85,B 0,C 180,E1 35293.855,E2 35293.855} C_VEL
LIN {X 0,Y 120.331,Z 740.348,A -85,B 0,C 180,E1 35292.881,E2 35292.881} C_VEL
LIN {X 0,Y 126.387,Z 737.731,A -85,B 0,C 180,E1 35293.575,E2 35293.575} C_VEL
LIN {X 0,Y 131.584,Z 754.988,A -85,B 0,C 180,E1 35339.466,E2 35339.466} C_VEL
LIN {X 0,Y 161.521,Z 760.175,A -85,B 0,C 180,E1 35359.571,E2 35359.571} C_VEL
LIN {X 0,Y 174.121,Z 761.197,A -85,B 0,C 180,E1 35368.096,E2 35368.096} C_VEL
LIN {X 0,Y 173.28,Z 761.173,A -85,B 0,C 180,E1 35372.508,E2 35372.508} C_VEL
LIN {X 0,Y 154.834,Z 759.382,A -85,B 0,C 180,E1 35384.174,E2 35384.174} C_VEL
LIN {X 0,Y 118.68,Z 749.329,A -85,B 0,C 180,E1 35419.412,E2 35419.412} C_VEL
LIN {X 0,Y 126.207,Z 737.805,A -85,B 0,C 180,E1 35446.464,E2 35446.464} C_VEL
LIN {X 0,Y 64.05,Z 758.096,A -85,B 0,C 180,E1 35446.436,E2 35446.436} C_VEL
LIN {X 0,Y 9.404,Z 764.805,A -85,B 0,C 180,E1 35423.741,E2 35423.741} C_VEL
LIN {X 0,Y 39.24,Z 762.41,A -85,B 0,C 180,E1 35294.952,E2 35294.952} C_VEL
LIN {X 0,Y 55.897,Z 759.774,A -85,B 0,C 180,E1 35293.855,E2 35293.855} C_VEL
LIN {X 0,Y 90.093,Z 751.829,A -85,B 0,C 180,E1 35298.155,E2 35298.155} C_VEL
LIN {X 0,Y 115.435,Z 743.068,A -85,B 0,C 180,E1 35297.478,E2 35297.478} C_VEL
LIN {X 0,Y 136.586,Z 758.647,A -85,B 0,C 180,E1 35350.197,E2 35350.197} C_VEL
LIN {X 0,Y 159.673,Z 761.216,A -85,B 0,C 180,E1 35364.19,E2 35364.19} C_VEL
LIN {X 0,Y 166.032,Z 761.504,A -85,B 0,C 180,E1 35370,E2 35370} C_VEL
LIN {X 0,Y 155.372,Z 760.846,A -85,B 0,C 180,E1 35378.419,E2 35378.419} C_VEL
LIN {X 0,Y 126.737,Z 757.122,A -85,B 0,C 180,E1 35396.586,E2 35396.586} C_VEL
LIN {X 0,Y 115.194,Z 743.167,A -85,B 0,C 180,E1 35442.485,E2 35442.485} C_VEL
LIN {X 0,Y 57.186,Z 759.85,A -85,B 0,C 180,E1 35438.149,E2 35438.149} C_VEL
LIN {X 0,Y 15.576,Z 764.631,A -85,B 0,C 180,E1 35399.133,E2 35399.133} C_VEL
LIN {X 0,Y 42.085,Z 762.235,A -85,B 0,C 180,E1 35305.734,E2 35305.734} C_VEL
LIN {X 0,Y 90.093,Z 751.829,A -85,B 0,C 180,E1 35298.155,E2 35298.155} C_VEL
LIN {X 0,Y 98.598,Z 750.086,A -85,B 0,C 180,E1 35303.242,E2 35303.242} C_VEL
LIN {X 0,Y 102.823,Z 752.047,A -85,B 0,C 180,E1 35316.67,E2 35316.67} C_VEL
LIN {X 0,Y 133.459,Z 760.094,A -85,B 0,C 180,E1 35354.346,E2 35354.346} C_VEL
LIN {X 0,Y 154.786,Z 761.577,A -85,B 0,C 180,E1 35367.192,E2 35367.192} C_VEL
LIN {X 0,Y 158.041,Z 761.679,A -85,B 0,C 180,E1 35370,E2 35370} C_VEL
LIN {X 0,Y 144.391,Z 761.09,A -85,B 0,C 180,E1 35379.064,E2 35379.064} C_VEL
LIN {X 0,Y 106.8,Z 755.366,A -85,B 0,C 180,E1 35409.716,E2 35409.716} C_VEL
LIN {X 0,Y 104.998,Z 747.767,A -85,B 0,C 180,E1 35437.99,E2 35437.99} C_VEL
LIN {X 0,Y 46.187,Z 762.06,A -85,B 0,C 180,E1 35425.171,E2 35425.171} C_VEL
LIN {X 0,Y 22.873,Z 764.458,A -85,B 0,C 180,E1 35350.642,E2 35350.642} C_VEL
LIN {X 0,Y 79.406,Z 755.448,A -85,B 0,C 180,E1 35304.886,E2 35304.886} C_VEL
LIN {X 0,Y 104.864,Z 747.966,A -85,B 0,C 180,E1 35302.822,E2 35302.822} C_VEL
LIN {X 0,Y 102.823,Z 752.047,A -85,B 0,C 180,E1 35316.67,E2 35316.67} C_VEL
LIN {X 0,Y 102.751,Z 757.632,A -85,B 0,C 180,E1 35336.209,E2 35336.209} C_VEL
LIN {X 0,Y 133.085,Z 761.338,A -85,B 0,C 180,E1 35360.159,E2 35360.159} C_VEL
LIN {X 0,Y 149.227,Z 761.871,A -85,B 0,C 180,E1 35370,E2 35370} C_VEL
LIN {X 0,Y 130.875,Z 761.217,A -85,B 0,C 180,E1 35380.912,E2 35380.912} C_VEL
LIN {X 0,Y 95.216,Z 752.134,A -85,B 0,C 180,E1 35431.161,E2 35431.161} C_VEL
LIN {X 0,Y 51.278,Z 761.885,A -85,B 0,C 180,E1 35417.676,E2 35417.676} C_VEL
LIN {X 0,Y 30.603,Z 764.283,A -85,B 0,C 180,E1 35355.656,E2 35355.656} C_VEL
LIN {X 0,Y 83.173,Z 755.271,A -85,B 0,C 180,E1 35309.997,E2 35309.997} C_VEL
LIN {X 0,Y 94.263,Z 752.178,A -85,B 0,C 180,E1 35307.77,E2 35307.77} C_VEL
LIN {X 0,Y 102.751,Z 757.632,A -85,B 0,C 180,E1 35336.209,E2 35336.209} C_VEL
LIN {X 0,Y 113.216,Z 761.06,A -85,B 0,C 180,E1 35354.288,E2 35354.288} C_VEL
LIN {X 0,Y 139.782,Z 762.078,A -85,B 0,C 180,E1 35370,E2 35370} C_VEL
LIN {X 0,Y 116.483,Z 761.36,A -85,B 0,C 180,E1 35383.347,E2 35383.347} C_VEL
LIN {X 0,Y 86.952,Z 755.46,A -85,B 0,C 180,E1 35424.266,E2 35424.266} C_VEL
LIN {X 0,Y 45.988,Z 763.301,A -85,B 0,C 180,E1 35399.647,E2 35399.647} C_VEL
LIN {X 0,Y 38.487,Z 764.108,A -85,B 0,C 180,E1 35358.639,E2 35358.639} C_VEL
LIN {X 0,Y 83.983,Z 756.098,A -85,B 0,C 180,E1 35315.654,E2 35315.654} C_VEL
LIN {X 0,Y 87.273,Z 755.68,A -85,B 0,C 180,E1 35317.103,E2 35317.103} C_VEL
LIN {X 0,Y 113.216,Z 761.06,A -85,B 0,C 180,E1 35354.288,E2 35354.288} C_VEL
LIN {X 0,Y 121.213,Z 762.231,A -85,B 0,C 180,E1 35365.31,E2 35365.31} C_VEL
LIN {X 0,Y 128.516,Z 762.3,A -85,B 0,C 180,E1 35370.608,E2 35370.608} C_VEL
LIN {X 0,Y 92.841,Z 760.806,A -85,B 0,C 180,E1 35394.102,E2 35394.102} C_VEL
LIN {X 0,Y 80.278,Z 758.202,A -85,B 0,C 180,E1 35415.701,E2 35415.701} C_VEL
LIN {X 0,Y 46.51,Z 763.932,A -85,B 0,C 180,E1 35379.384,E2 35379.384} C_VEL
LIN {X 0,Y 63.43,Z 761.535,A -85,B 0,C 180,E1 35333.295,E2 35333.295} C_VEL
LIN {X 0,Y 80.605,Z 758.14,A -85,B 0,C 180,E1 35324.251,E2 35324.251} C_VEL
LIN {X 0,Y 121.213,Z 762.231,A -85,B 0,C 180,E1 35365.31,E2 35365.31} C_VEL
LIN {X 0,Y 118.862,Z 762.533,A -85,B 0,C 180,E1 35370.162,E2 35370.162} C_VEL
LIN {X 0,Y 108.468,Z 762.484,A -85,B 0,C 180,E1 35375.434,E2 35375.434} C_VEL
LIN {X 0,Y 75.544,Z 760.349,A -85,B 0,C 180,E1 35406.133,E2 35406.133} C_VEL
LIN {X 0,Y 54.472,Z 763.757,A -85,B 0,C 180,E1 35378.002,E2 35378.002} C_VEL
LIN {X 0,Y 72.129,Z 760.94,A -85,B 0,C 180,E1 35335.639,E2 35335.639} C_VEL
LIN {X 0,Y 75.964,Z 760.309,A -85,B 0,C 180,E1 35333.892,E2 35333.892} C_VEL
LIN {X 0,Y 117.892,Z 762.527,A -85,B 0,C 180,E1 35369.231,E2 35369.231} C_VEL
LIN {X 0,Y 108.468,Z 762.484,A -85,B 0,C 180,E1 35375.434,E2 35375.434} C_VEL
LIN {X 0,Y 79.669,Z 762.354,A -85,B 0,C 180,E1 35388.12,E2 35388.12} C_VEL
LIN {X 0,Y 73.507,Z 761.998,A -85,B 0,C 180,E1 35395.05,E2 35395.05} C_VEL
LIN {X 0,Y 62.446,Z 763.583,A -85,B 0,C 180,E1 35363.026,E2 35363.026} C_VEL
LIN {X 0,Y 74.475,Z 762.002,A -85,B 0,C 180,E1 35345.595,E2 35345.595} C_VEL
LIN {X 0,Y 107.86,Z 762.775,A -85,B 0,C 180,E1 35369.903,E2 35369.903} C_VEL
LIN {X 0,Y 79.669,Z 762.354,A -85,B 0,C 180,E1 35388.12,E2 35388.12} C_VEL
LIN {X 0,Y 72.03,Z 763.164,A -85,B 0,C 180,E1 35382.694,E2 35382.694} C_VEL
LIN {X 0,Y 70.102,Z 763.407,A -85,B 0,C 180,E1 35371.256,E2 35371.256} C_VEL
LIN {X 0,Y 75.349,Z 763.018,A -85,B 0,C 180,E1 35356.76,E2 35356.76} C_VEL
LIN {X 0,Y 95.287,Z 763.05,A -85,B 0,C 180,E1 35370,E2 35370} C_VEL
LIN {X 0,Y 74.621,Z 763.035,A -85,B 0,C 180,E1 35383.372,E2 35383.372} C_VEL
LIN {X 0,Y 70.102,Z 763.407,A -85,B 0,C 180,E1 35371.256,E2 35371.256} C_VEL
LIN {X 0,Y 81.654,Z 763.352,A -85,B 0,C 180,E1 35369.247,E2 35369.247} C_VEL
LIN {X 0,Y 82.387,Z 763.332,A -85,B 0,C 180,E1 35369.997,E2 35369.997} C_VEL
LIN {X 0,Y 79.19,Z 763.352,A -85,B 0,C 180,E1 35371.789,E2 35371.789} C_VEL
LIN {X 0,Y 80.259,Z 763.336,A -85,B 0,C 180,E1 35368.463,E2 35368.463} C_VEL
LIN {X 0,Y 82.387,Z 763.332,A -85,B 0,C 180,E1 35369.997,E2 35369.997} C_VEL
LIN {X 0,Y 83.817,Z 765.332,A -85,B 0,C 180,E1 35370.963,E2 35370.963} C_VEL
LIN {X 0,Y 83.817,Z 783.5,A -85,B 0,C 180,E1 35370.963,E2 35370.963} C_VEL
LIN {X 0,Y 83.817,Z 783.5,A -85,B 0,C 180,E1 35370.963,E2 35370.963}

QRS_NEXT_CUT()
PTP {E1 35457.084,E2 35457.084}
PTP {X 0,Y 759.931,A -85,B 0,C 180,E1 35457.084,E2 35457.084,E3 0,E4 0,E5 0,E6 0}
QRS_SPEED_INIT()
LIN {X 0,Y 759.931,Z 783.5,A -85,B 0,C 180,E1 35457.084,E2 35457.084,E3 0,E4 0,E5 0,E6 0} C_VEL
LIN {X 0,Y 759.931,Z 176.589,A -85,B 0,C 180,E1 35457.084,E2 35457.084} C_VEL
LIN {X 0,Y 759.931,Z 168.515,A -85,B 0,C 180,E1 35457.084,E2 35457.084} C_VEL
LIN {X 0,Y 759.9,Z 166.515,A -85,B 0,C 180,E1 35456.933,E2 35456.933} C_VEL
LIN {X 0,Y 759.811,Z 166.515,A -85,B 0,C 180,E1 35454.26,E2 35454.26} C_VEL
LIN {X 0,Y 759.808,Z 166.514,A -85,B 0,C 180,E1 35452.058,E2 35452.058} C_VEL
LIN {X 0,Y 759.821,Z 166.515,A -85,B 0,C 180,E1 35449.767,E2 35449.767} C_VEL
LIN {X 0,Y 759.876,Z 166.515,A -85,B 0,C 180,E1 35446.919,E2 35446.919} C_VEL
LIN {X 0,Y 759.81,Z 166.515,A -85,B 0,C 180,E1 35444.349,E2 35444.349} C_VEL
LIN {X 0,Y 759.81,Z 166.515,A -85,B 0,C 180,E1 35442.049,E2 35442.049} C_VEL
LIN {X 0,Y 759.842,Z 166.515,A -85,B 0,C 180,E1 35439.671,E2 35439.671} C_VEL
LIN {X 0,Y 759.83,Z 166.515,A -85,B 0,C 180,E1 35436.693,E2 35436.693} C_VEL
LIN {X 0,Y 759.808,Z 166.514,A -85,B 0,C 180,E1 35434.332,E2 35434.332} C_VEL
LIN {X 0,Y 759.814,Z 166.513,A -85,B 0,C 180,E1 35432.064,E2 35432.064} C_VEL
LIN {X 0,Y 759.906,Z 166.516,A -85,B 0,C 180,E1 35429.3,E2 35429.3} C_VEL
LIN {X 0,Y 759.815,Z 166.515,A -85,B 0,C 180,E1 35426.628,E2 35426.628} C_VEL
LIN {X 0,Y 759.805,Z 166.514,A -85,B 0,C 180,E1 35424.406,E2 35424.406} C_VEL
LIN {X 0,Y 759.813,Z 166.515,A -85,B 0,C 180,E1 35422.176,E2 35422.176} C_VEL
LIN {X 0,Y 759.907,Z 166.515,A -85,B 0,C 180,E1 35419.386,E2 35419.386} C_VEL
LIN {X 0,Y 759.812,Z 166.515,A -85,B 0,C 180,E1 35416.688,E2 35416.688} C_VEL
LIN {X 0,Y 759.808,Z 166.515,A -85,B 0,C 180,E1 35414.391,E2 35414.391} C_VEL
LIN {X 0,Y 759.834,Z 166.515,A -85,B 0,C 180,E1 35412.045,E2 35412.045} C_VEL
LIN {X 0,Y 759.836,Z 166.515,A -85,B 0,C 180,E1 35409.068,E2 35409.068} C_VEL
LIN {X 0,Y 759.808,Z 166.515,A -85,B 0,C 180,E1 35406.682,E2 35406.682} C_VEL
LIN {X 0,Y 759.814,Z 166.515,A -85,B 0,C 180,E1 35404.366,E2 35404.366} C_VEL
LIN {X 0,Y 759.905,Z 166.515,A -85,B 0,C 180,E1 35401.575,E2 35401.575} C_VEL
LIN {X 0,Y 759.811,Z 166.515,A -85,B 0,C 180,E1 35398.875,E2 35398.875} C_VEL
LIN {X 0,Y 759.809,Z 166.515,A -85,B 0,C 180,E1 35396.575,E2 35396.575} C_VEL
LIN {X 0,Y 759.844,Z 166.515,A -85,B 0,C 180,E1 35394.154,E2 35394.154} C_VEL
LIN {X 0,Y 759.83,Z 166.515,A -85,B 0,C 180,E1 35391.213,E2 35391.213} C_VEL
LIN {X 0,Y 759.808,Z 166.515,A -85,B 0,C 180,E1 35388.881,E2 35388.881} C_VEL
LIN {X 0,Y 759.81,Z 166.515,A -85,B 0,C 180,E1 35386.658,E2 35386.658} C_VEL
LIN {X 0,Y 759.885,Z 166.515,A -85,B 0,C 180,E1 35384.009,E2 35384.009} C_VEL
LIN {X 0,Y 759.821,Z 166.515,A -85,B 0,C 180,E1 35381.229,E2 35381.229} C_VEL
LIN {X 0,Y 759.807,Z 166.515,A -85,B 0,C 180,E1 35378.932,E2 35378.932} C_VEL
LIN {X 0,Y 759.811,Z 166.515,A -85,B 0,C 180,E1 35376.725,E2 35376.725} C_VEL
LIN {X 0,Y 759.91,Z 166.515,A -85,B 0,C 180,E1 35373.998,E2 35373.998} C_VEL
LIN {X 0,Y 759.816,Z 166.515,A -85,B 0,C 180,E1 35371.282,E2 35371.282} C_VEL
LIN {X 0,Y 759.806,Z 166.515,A -85,B 0,C 180,E1 35369.095,E2 35369.095} C_VEL
LIN {X 0,Y 759.807,Z 166.515,A -85,B 0,C 180,E1 35366.908,E2 35366.908} C_VEL
LIN {X 0,Y 759.844,Z 166.515,A -85,B 0,C 180,E1 35364.488,E2 35364.488} C_VEL
LIN {X 0,Y 759.828,Z 166.515,A -85,B 0,C 180,E1 35361.526,E2 35361.526} C_VEL
LIN {X 0,Y 759.807,Z 166.515,A -85,B 0,C 180,E1 35359.155,E2 35359.155} C_VEL
LIN {X 0,Y 759.816,Z 166.515,A -85,B 0,C 180,E1 35356.86,E2 35356.86} C_VEL
LIN {X 0,Y 759.891,Z 166.515,A -85,B 0,C 180,E1 35354.04,E2 35354.04} C_VEL
LIN {X 0,Y 759.813,Z 166.515,A -85,B 0,C 180,E1 35351.433,E2 35351.433} C_VEL
LIN {X 0,Y 759.807,Z 166.515,A -85,B 0,C 180,E1 35349.271,E2 35349.271} C_VEL
LIN {X 0,Y 759.815,Z 166.515,A -85,B 0,C 180,E1 35346.996,E2 35346.996} C_VEL
LIN {X 0,Y 759.914,Z 166.515,A -85,B 0,C 180,E1 35344.269,E2 35344.269} C_VEL
LIN {X 0,Y 759.812,Z 166.515,A -85,B 0,C 180,E1 35341.531,E2 35341.531} C_VEL
LIN {X 0,Y 759.806,Z 166.515,A -85,B 0,C 180,E1 35339.301,E2 35339.301} C_VEL
LIN {X 0,Y 759.842,Z 166.515,A -85,B 0,C 180,E1 35336.817,E2 35336.817} C_VEL
LIN {X 0,Y 759.833,Z 166.515,A -85,B 0,C 180,E1 35333.882,E2 35333.882} C_VEL
LIN {X 0,Y 759.808,Z 166.515,A -85,B 0,C 180,E1 35331.51,E2 35331.51} C_VEL
LIN {X 0,Y 759.812,Z 166.515,A -85,B 0,C 180,E1 35329.26,E2 35329.26} C_VEL
LIN {X 0,Y 759.899,Z 166.515,A -85,B 0,C 180,E1 35326.58,E2 35326.58} C_VEL
LIN {X 0,Y 759.817,Z 166.515,A -85,B 0,C 180,E1 35323.804,E2 35323.804} C_VEL
LIN {X 0,Y 759.807,Z 166.515,A -85,B 0,C 180,E1 35321.549,E2 35321.549} C_VEL
LIN {X 0,Y 759.817,Z 166.515,A -85,B 0,C 180,E1 35319.27,E2 35319.27} C_VEL
LIN {X 0,Y 759.896,Z 166.514,A -85,B 0,C 180,E1 35316.495,E2 35316.495} C_VEL
LIN {X 0,Y 759.814,Z 166.514,A -85,B 0,C 180,E1 35313.874,E2 35313.874} C_VEL
LIN {X 0,Y 759.808,Z 166.515,A -85,B 0,C 180,E1 35311.585,E2 35311.585} C_VEL
LIN {X 0,Y 759.827,Z 166.515,A -85,B 0,C 180,E1 35309.267,E2 35309.267} C_VEL
LIN {X 0,Y 759.85,Z 166.514,A -85,B 0,C 180,E1 35306.325,E2 35306.325} C_VEL
LIN {X 0,Y 759.809,Z 166.515,A -85,B 0,C 180,E1 35303.829,E2 35303.829} C_VEL
LIN {X 0,Y 759.814,Z 166.515,A -85,B 0,C 180,E1 35301.525,E2 35301.525} C_VEL
LIN {X 0,Y 759.918,Z 166.515,A -85,B 0,C 180,E1 35298.806,E2 35298.806} C_VEL
LIN {X 0,Y 759.812,Z 166.515,A -85,B 0,C 180,E1 35296.043,E2 35296.043} C_VEL
LIN {X 0,Y 759.807,Z 166.515,A -85,B 0,C 180,E1 35293.818,E2 35293.818} C_VEL
LIN {X 0,Y 759.833,Z 166.514,A -85,B 0,C 180,E1 35291.41,E2 35291.41} C_VEL
LIN {X 0,Y 759.835,Z 166.514,A -85,B 0,C 180,E1 35288.399,E2 35288.399} C_VEL
LIN {X 0,Y 759.808,Z 166.515,A -85,B 0,C 180,E1 35286.043,E2 35286.043} C_VEL
LIN {X 0,Y 759.809,Z 166.515,A -85,B 0,C 180,E1 35283.848,E2 35283.848} C_VEL
LIN {X 0,Y 759.843,Z 166.514,A -85,B 0,C 180,E1 35281.433,E2 35281.433} C_VEL
LIN {X 0,Y 759.832,Z 166.514,A -85,B 0,C 180,E1 35278.492,E2 35278.492} C_VEL
LIN {X 0,Y 759.809,Z 166.515,A -85,B 0,C 180,E1 35276.152,E2 35276.152} C_VEL
LIN {X 0,Y 759.812,Z 166.515,A -85,B 0,C 180,E1 35273.881,E2 35273.881} C_VEL
LIN {X 0,Y 759.882,Z 166.514,A -85,B 0,C 180,E1 35271.296,E2 35271.296} C_VEL
LIN {X 0,Y 759.82,Z 166.514,A -85,B 0,C 180,E1 35268.461,E2 35268.461} C_VEL
LIN {X 0,Y 759.808,Z 166.515,A -85,B 0,C 180,E1 35266.142,E2 35266.142} C_VEL
LIN {X 0,Y 759.822,Z 166.515,A -85,B 0,C 180,E1 35263.845,E2 35263.845} C_VEL
LIN {X 0,Y 759.882,Z 166.515,A -85,B 0,C 180,E1 35261.033,E2 35261.033} C_VEL
LIN {X 0,Y 759.813,Z 166.514,A -85,B 0,C 180,E1 35258.46,E2 35258.46} C_VEL
LIN {X 0,Y 759.81,Z 166.515,A -85,B 0,C 180,E1 35256.171,E2 35256.171} C_VEL
LIN {X 0,Y 759.866,Z 166.515,A -85,B 0,C 180,E1 35253.591,E2 35253.591} C_VEL
LIN {X 0,Y 759.826,Z 166.514,A -85,B 0,C 180,E1 35250.733,E2 35250.733} C_VEL
LIN {X 0,Y 759.811,Z 166.515,A -85,B 0,C 180,E1 35248.499,E2 35248.499} C_VEL
LIN {X 0,Y 759.814,Z 166.515,A -85,B 0,C 180,E1 35246.175,E2 35246.175} C_VEL
LIN {X 0,Y 759.904,Z 166.514,A -85,B 0,C 180,E1 35243.499,E2 35243.499} C_VEL
LIN {X 0,Y 759.818,Z 166.514,A -85,B 0,C 180,E1 35240.73,E2 35240.73} C_VEL
LIN {X 0,Y 759.809,Z 166.515,A -85,B 0,C 180,E1 35238.451,E2 35238.451} C_VEL
LIN {X 0,Y 759.823,Z 166.515,A -85,B 0,C 180,E1 35236.141,E2 35236.141} C_VEL
LIN {X 0,Y 759.871,Z 166.514,A -85,B 0,C 180,E1 35233.273,E2 35233.273} C_VEL
LIN {X 0,Y 759.812,Z 166.515,A -85,B 0,C 180,E1 35230.711,E2 35230.711} C_VEL
LIN {X 0,Y 759.811,Z 166.514,A -85,B 0,C 180,E1 35228.463,E2 35228.463} C_VEL
LIN {X 0,Y 759.855,Z 166.514,A -85,B 0,C 180,E1 35225.974,E2 35225.974} C_VEL
LIN {X 0,Y 759.827,Z 166.514,A -85,B 0,C 180,E1 35223.043,E2 35223.043} C_VEL
LIN {X 0,Y 759.809,Z 166.515,A -85,B 0,C 180,E1 35220.699,E2 35220.699} C_VEL
LIN {X 0,Y 759.898,Z 166.828,A -85,B 0,C 180,E1 35219.784,E2 35219.784} C_VEL
LIN {X 0,Y 759.911,Z 201.036,A -85,B 0,C 180,E1 35217.191,E2 35217.191} C_VEL
LIN {X 0,Y 759.897,Z 226.466,A -85,B 0,C 180,E1 35215.335,E2 35215.335} C_VEL
LIN {X 0,Y 759.907,Z 485.76,A -85,B 0,C 180,E1 35212.698,E2 35212.698} C_VEL
LIN {X 0,Y 759.906,Z 531.263,A -85,B 0,C 180,E1 35212.215,E2 35212.215} C_VEL
LIN {X 0,Y 759.914,Z 552.968,A -85,B 0,C 180,E1 35211.838,E2 35211.838} C_VEL
LIN {X 0,Y 759.905,Z 573.872,A -85,B 0,C 180,E1 35211.344,E2 35211.344} C_VEL
LIN {X 0,Y 759.906,Z 593.193,A -85,B 0,C 180,E1 35210.767,E2 35210.767} C_VEL
LIN {X 0,Y 759.919,Z 612.949,A -85,B 0,C 180,E1 35210.036,E2 35210.036} C_VEL
LIN {X 0,Y 759.918,Z 632.609,A -85,B 0,C 180,E1 35209.169,E2 35209.169} C_VEL
LIN {X 0,Y 759.914,Z 651.31,A -85,B 0,C 180,E1 35208.193,E2 35208.193} C_VEL
LIN {X 0,Y 759.916,Z 669.112,A -85,B 0,C 180,E1 35207.1,E2 35207.1} C_VEL
LIN {X 0,Y 759.919,Z 686.23,A -85,B 0,C 180,E1 35205.878,E2 35205.878} C_VEL
LIN {X 0,Y 759.915,Z 701.339,A -85,B 0,C 180,E1 35204.631,E2 35204.631} C_VEL
LIN {X 0,Y 759.909,Z 715.893,A -85,B 0,C 180,E1 35203.233,E2 35203.233} C_VEL
LIN {X 0,Y 759.916,Z 728.193,A -85,B 0,C 180,E1 35201.843,E2 35201.843} C_VEL
LIN {X 0,Y 759.912,Z 739.779,A -85,B 0,C 180,E1 35200.307,E2 35200.307} C_VEL
LIN {X 0,Y 759.914,Z 749.437,A -85,B 0,C 180,E1 35198.778,E2 35198.778} C_VEL
LIN {X 0,Y 759.912,Z 757.529,A -85,B 0,C 180,E1 35197.18,E2 35197.18} C_VEL
LIN {X 0,Y 759.913,Z 764.148,A -85,B 0,C 180,E1 35195.511,E2 35195.511} C_VEL
LIN {X 0,Y 759.918,Z 768.827,A -85,B 0,C 180,E1 35193.923,E2 35193.923} C_VEL
LIN {X 0,Y 759.906,Z 771.895,A -85,B 0,C 180,E1 35192.262,E2 35192.262} C_VEL
LIN {X 0,Y 759.9,Z 773.33,A -85,B 0,C 180,E1 35190.603,E2 35190.603} C_VEL
LIN {X 0,Y 759.91,Z 773.209,A -85,B 0,C 180,E1 35189.02,E2 35189.02} C_VEL
LIN {X 0,Y 759.917,Z 771.337,A -85,B 0,C 180,E1 35187.361,E2 35187.361} C_VEL
LIN {X 0,Y 759.913,Z 767.808,A -85,B 0,C 180,E1 35185.699,E2 35185.699} C_VEL
LIN {X 0,Y 759.916,Z 762.875,A -85,B 0,C 180,E1 35184.11,E2 35184.11} C_VEL
LIN {X 0,Y 759.901,Z 756.116,A -85,B 0,C 180,E1 35182.516,E2 35182.516} C_VEL
LIN {X 0,Y 759.903,Z 747.599,A -85,B 0,C 180,E1 35180.916,E2 35180.916} C_VEL
LIN {X 0,Y 759.909,Z 737.696,A -85,B 0,C 180,E1 35179.386,E2 35179.386} C_VEL
LIN {X 0,Y 759.913,Z 726.274,A -85,B 0,C 180,E1 35177.926,E2 35177.926} C_VEL
LIN {X 0,Y 759.914,Z 712.793,A -85,B 0,C 180,E1 35176.457,E2 35176.457} C_VEL
LIN {X 0,Y 759.912,Z 698.679,A -85,B 0,C 180,E1 35175.135,E2 35175.135} C_VEL
LIN {X 0,Y 759.911,Z 682.735,A -85,B 0,C 180,E1 35173.85,E2 35173.85} C_VEL
LIN {X 0,Y 759.913,Z 665.492,A -85,B 0,C 180,E1 35172.663,E2 35172.663} C_VEL
LIN {X 0,Y 759.917,Z 647.416,A -85,B 0,C 180,E1 35171.594,E2 35171.594} C_VEL
LIN {X 0,Y 759.916,Z 628.499,A -85,B 0,C 180,E1 35170.635,E2 35170.635} C_VEL
LIN {X 0,Y 759.919,Z 608.82,A -85,B 0,C 180,E1 35169.797,E2 35169.797} C_VEL
LIN {X 0,Y 759.911,Z 589.067,A -85,B 0,C 180,E1 35169.103,E2 35169.103} C_VEL
LIN {X 0,Y 759.906,Z 568.527,A -85,B 0,C 180,E1 35168.513,E2 35168.513} C_VEL
LIN {X 0,Y 759.908,Z 546.731,A -85,B 0,C 180,E1 35168.04,E2 35168.04} C_VEL
LIN {X 0,Y 759.906,Z 525.817,A -85,B 0,C 180,E1 35167.718,E2 35167.718} C_VEL
LIN {X 0,Y 759.899,Z 245.791,A -85,B 0,C 180,E1 35164.871,E2 35164.871} C_VEL
LIN {X 0,Y 759.897,Z 226.183,A -85,B 0,C 180,E1 35164.654,E2 35164.654} C_VEL
LIN {X 0,Y 759.916,Z 189.489,A -85,B 0,C 180,E1 35161.944,E2 35161.944} C_VEL
LIN {X 0,Y 759.893,Z 166.664,A -85,B 0,C 180,E1 35160.188,E2 35160.188} C_VEL
LIN {X 0,Y 759.817,Z 166.514,A -85,B 0,C 180,E1 35157.621,E2 35157.621} C_VEL
LIN {X 0,Y 759.81,Z 166.515,A -85,B 0,C 180,E1 35155.268,E2 35155.268} C_VEL
LIN {X 0,Y 759.869,Z 166.514,A -85,B 0,C 180,E1 35152.661,E2 35152.661} C_VEL
LIN {X 0,Y 759.829,Z 166.515,A -85,B 0,C 180,E1 35149.855,E2 35149.855} C_VEL
LIN {X 0,Y 759.809,Z 166.515,A -85,B 0,C 180,E1 35147.546,E2 35147.546} C_VEL
LIN {X 0,Y 759.811,Z 166.515,A -85,B 0,C 180,E1 35145.361,E2 35145.361} C_VEL
LIN {X 0,Y 759.856,Z 166.514,A -85,B 0,C 180,E1 35142.869,E2 35142.869} C_VEL
LIN {X 0,Y 759.828,Z 166.514,A -85,B 0,C 180,E1 35139.955,E2 35139.955} C_VEL
LIN {X 0,Y 759.809,Z 166.515,A -85,B 0,C 180,E1 35137.617,E2 35137.617} C_VEL
LIN {X 0,Y 759.81,Z 166.514,A -85,B 0,C 180,E1 35135.464,E2 35135.464} C_VEL
LIN {X 0,Y 759.851,Z 166.514,A -85,B 0,C 180,E1 35133.01,E2 35133.01} C_VEL
LIN {X 0,Y 759.83,Z 166.514,A -85,B 0,C 180,E1 35130.091,E2 35130.091} C_VEL
LIN {X 0,Y 759.809,Z 166.514,A -85,B 0,C 180,E1 35127.766,E2 35127.766} C_VEL
LIN {X 0,Y 759.811,Z 166.514,A -85,B 0,C 180,E1 35125.572,E2 35125.572} C_VEL
LIN {X 0,Y 759.856,Z 166.515,A -85,B 0,C 180,E1 35123.088,E2 35123.088} C_VEL
LIN {X 0,Y 759.826,Z 166.515,A -85,B 0,C 180,E1 35120.168,E2 35120.168} C_VEL
LIN {X 0,Y 759.809,Z 166.514,A -85,B 0,C 180,E1 35117.856,E2 35117.856} C_VEL
LIN {X 0,Y 759.815,Z 166.515,A -85,B 0,C 180,E1 35115.573,E2 35115.573} C_VEL
LIN {X 0,Y 759.907,Z 166.516,A -85,B 0,C 180,E1 35112.848,E2 35112.848} C_VEL
LIN {X 0,Y 759.817,Z 166.515,A -85,B 0,C 180,E1 35110.157,E2 35110.157} C_VEL
LIN {X 0,Y 759.808,Z 166.514,A -85,B 0,C 180,E1 35107.866,E2 35107.866} C_VEL
LIN {X 0,Y 759.821,Z 166.515,A -85,B 0,C 180,E1 35105.588,E2 35105.588} C_VEL
LIN {X 0,Y 759.872,Z 166.515,A -85,B 0,C 180,E1 35102.715,E2 35102.715} C_VEL
LIN {X 0,Y 759.814,Z 166.515,A -85,B 0,C 180,E1 35100.226,E2 35100.226} C_VEL
LIN {X 0,Y 759.807,Z 166.514,A -85,B 0,C 180,E1 35098.039,E2 35098.039} C_VEL
LIN {X 0,Y 759.9,Z 166.515,A -85,B 0,C 180,E1 35096.933,E2 35096.933} C_VEL
LIN {X 0,Y 758.844,Z 166.638,A -85,B 0,C 180,E1 35096.353,E2 35096.353} C_VEL
LIN {X 0,Y 752.418,Z 167.444,A -85,B 0,C 180,E1 35094.727,E2 35094.727} C_VEL
LIN {X 0,Y 751.875,Z 167.504,A -85,B 0,C 180,E1 35094.304,E2 35094.304} C_VEL
LIN {X 0,Y 751.869,Z 167.503,A -85,B 0,C 180,E1 35092.05,E2 35092.05} C_VEL
LIN {X 0,Y 751.886,Z 167.504,A -85,B 0,C 180,E1 35089.72,E2 35089.72} C_VEL
LIN {X 0,Y 751.914,Z 167.504,A -85,B 0,C 180,E1 35086.778,E2 35086.778} C_VEL
LIN {X 0,Y 751.871,Z 167.504,A -85,B 0,C 180,E1 35084.3,E2 35084.3} C_VEL
LIN {X 0,Y 751.876,Z 167.503,A -85,B 0,C 180,E1 35081.949,E2 35081.949} C_VEL
LIN {X 0,Y 751.968,Z 167.504,A -85,B 0,C 180,E1 35079.286,E2 35079.286} C_VEL
LIN {X 0,Y 751.88,Z 167.504,A -85,B 0,C 180,E1 35076.559,E2 35076.559} C_VEL
LIN {X 0,Y 751.869,Z 167.503,A -85,B 0,C 180,E1 35074.223,E2 35074.223} C_VEL
LIN {X 0,Y 751.894,Z 167.5,A -85,B 0,C 180,E1 35071.83,E2 35071.83} C_VEL
LIN {X 0,Y 751.898,Z 167.504,A -85,B 0,C 180,E1 35068.848,E2 35068.848} C_VEL
LIN {X 0,Y 751.869,Z 167.503,A -85,B 0,C 180,E1 35066.411,E2 35066.411} C_VEL
LIN {X 0,Y 751.872,Z 167.502,A -85,B 0,C 180,E1 35064.187,E2 35064.187} C_VEL
LIN {X 0,Y 751.961,Z 167.504,A -85,B 0,C 180,E1 35061.515,E2 35061.515} C_VEL
LIN {X 0,Y 751.877,Z 167.504,A -85,B 0,C 180,E1 35058.73,E2 35058.73} C_VEL
LIN {X 0,Y 751.869,Z 167.504,A -85,B 0,C 180,E1 35056.442,E2 35056.442} C_VEL
LIN {X 0,Y 751.897,Z 167.504,A -85,B 0,C 180,E1 35053.992,E2 35053.992} C_VEL
LIN {X 0,Y 751.899,Z 167.504,A -85,B 0,C 180,E1 35051.059,E2 35051.059} C_VEL
LIN {X 0,Y 751.87,Z 167.504,A -85,B 0,C 180,E1 35048.679,E2 35048.679} C_VEL
LIN {X 0,Y 751.872,Z 167.504,A -85,B 0,C 180,E1 35046.431,E2 35046.431} C_VEL
LIN {X 0,Y 751.951,Z 167.504,A -85,B 0,C 180,E1 35043.762,E2 35043.762} C_VEL
LIN {X 0,Y 751.877,Z 167.504,A -85,B 0,C 180,E1 35040.934,E2 35040.934} C_VEL
LIN {X 0,Y 751.869,Z 167.504,A -85,B 0,C 180,E1 35038.687,E2 35038.687} C_VEL
LIN {X 0,Y 751.889,Z 167.504,A -85,B 0,C 180,E1 35036.281,E2 35036.281} C_VEL
LIN {X 0,Y 751.895,Z 167.504,A -85,B 0,C 180,E1 35033.232,E2 35033.232} C_VEL
LIN {X 0,Y 751.87,Z 167.504,A -85,B 0,C 180,E1 35030.877,E2 35030.877} C_VEL
LIN {X 0,Y 751.873,Z 167.504,A -85,B 0,C 180,E1 35028.61,E2 35028.61} C_VEL
LIN {X 0,Y 751.964,Z 167.504,A -85,B 0,C 180,E1 35025.895,E2 35025.895} C_VEL
LIN {X 0,Y 751.878,Z 167.504,A -85,B 0,C 180,E1 35023.143,E2 35023.143} C_VEL
LIN {X 0,Y 751.868,Z 167.504,A -85,B 0,C 180,E1 35020.884,E2 35020.884} C_VEL
LIN {X 0,Y 751.888,Z 167.504,A -85,B 0,C 180,E1 35018.487,E2 35018.487} C_VEL
LIN {X 0,Y 751.903,Z 167.504,A -85,B 0,C 180,E1 35015.494,E2 35015.494} C_VEL
LIN {X 0,Y 751.869,Z 167.505,A -85,B 0,C 180,E1 35013.125,E2 35013.125} C_VEL
LIN {X 0,Y 751.869,Z 167.504,A -85,B 0,C 180,E1 35010.914,E2 35010.914} C_VEL
LIN {X 0,Y 751.884,Z 167.504,A -85,B 0,C 180,E1 35008.629,E2 35008.629} C_VEL
LIN {X 0,Y 751.92,Z 167.504,A -85,B 0,C 180,E1 35005.73,E2 35005.73} C_VEL
LIN {X 0,Y 751.87,Z 167.504,A -85,B 0,C 180,E1 35003.204,E2 35003.204} C_VEL
LIN {X 0,Y 751.87,Z 167.504,A -85,B 0,C 180,E1 35000.973,E2 35000.973} C_VEL
LIN {X 0,Y 751.925,Z 167.504,A -85,B 0,C 180,E1 34998.418,E2 34998.418} C_VEL
LIN {X 0,Y 751.884,Z 167.504,A -85,B 0,C 180,E1 34995.524,E2 34995.524} C_VEL
LIN {X 0,Y 751.868,Z 167.504,A -85,B 0,C 180,E1 34993.229,E2 34993.229} C_VEL
LIN {X 0,Y 751.879,Z 167.504,A -85,B 0,C 180,E1 34990.907,E2 34990.907} C_VEL
LIN {X 0,Y 751.96,Z 167.504,A -85,B 0,C 180,E1 34988.144,E2 34988.144} C_VEL
LIN {X 0,Y 751.873,Z 167.504,A -85,B 0,C 180,E1 34985.455,E2 34985.455} C_VEL
LIN {X 0,Y 751.871,Z 167.504,A -85,B 0,C 180,E1 34983.17,E2 34983.17} C_VEL
LIN {X 0,Y 751.939,Z 167.504,A -85,B 0,C 180,E1 34980.532,E2 34980.532} C_VEL
LIN {X 0,Y 751.88,Z 167.504,A -85,B 0,C 180,E1 34977.688,E2 34977.688} C_VEL
LIN {X 0,Y 751.869,Z 167.504,A -85,B 0,C 180,E1 34975.312,E2 34975.312} C_VEL
LIN {X 0,Y 751.915,Z 167.504,A -85,B 0,C 180,E1 34972.773,E2 34972.773} C_VEL
LIN {X 0,Y 751.886,Z 167.504,A -85,B 0,C 180,E1 34969.843,E2 34969.843} C_VEL
LIN {X 0,Y 751.868,Z 167.504,A -85,B 0,C 180,E1 34967.508,E2 34967.508} C_VEL
LIN {X 0,Y 751.875,Z 167.504,A -85,B 0,C 180,E1 34965.247,E2 34965.247} C_VEL
LIN {X 0,Y 751.965,Z 167.505,A -85,B 0,C 180,E1 34962.492,E2 34962.492} C_VEL
LIN {X 0,Y 751.874,Z 167.504,A -85,B 0,C 180,E1 34959.767,E2 34959.767} C_VEL
LIN {X 0,Y 751.871,Z 167.504,A -85,B 0,C 180,E1 34957.427,E2 34957.427} C_VEL
LIN {X 0,Y 751.913,Z 167.502,A -85,B 0,C 180,E1 34954.97,E2 34954.97} C_VEL
LIN {X 0,Y 751.887,Z 167.504,A -85,B 0,C 180,E1 34952.047,E2 34952.047} C_VEL
LIN {X 0,Y 751.87,Z 167.503,A -85,B 0,C 180,E1 34949.739,E2 34949.739} C_VEL
LIN {X 0,Y 751.874,Z 167.5,A -85,B 0,C 180,E1 34947.482,E2 34947.482} C_VEL
LIN {X 0,Y 751.962,Z 167.505,A -85,B 0,C 180,E1 34944.761,E2 34944.761} C_VEL
LIN {X 0,Y 751.877,Z 167.503,A -85,B 0,C 180,E1 34942.026,E2 34942.026} C_VEL
LIN {X 0,Y 751.87,Z 167.504,A -85,B 0,C 180,E1 34939.709,E2 34939.709} C_VEL
LIN {X 0,Y 751.887,Z 167.503,A -85,B 0,C 180,E1 34937.41,E2 34937.41} C_VEL
LIN {X 0,Y 751.912,Z 167.504,A -85,B 0,C 180,E1 34934.478,E2 34934.478} C_VEL
LIN {X 0,Y 751.87,Z 167.503,A -85,B 0,C 180,E1 34931.974,E2 34931.974} C_VEL
LIN {X 0,Y 751.877,Z 167.504,A -85,B 0,C 180,E1 34929.646,E2 34929.646} C_VEL
LIN {X 0,Y 751.969,Z 167.503,A -85,B 0,C 180,E1 34926.873,E2 34926.873} C_VEL
LIN {X 0,Y 751.874,Z 167.504,A -85,B 0,C 180,E1 34924.194,E2 34924.194} C_VEL
LIN {X 0,Y 751.87,Z 167.503,A -85,B 0,C 180,E1 34921.905,E2 34921.905} C_VEL
LIN {X 0,Y 751.894,Z 167.504,A -85,B 0,C 180,E1 34919.543,E2 34919.543} C_VEL
LIN {X 0,Y 751.892,Z 167.503,A -85,B 0,C 180,E1 34916.493,E2 34916.493} C_VEL
LIN {X 0,Y 751.87,Z 167.504,A -85,B 0,C 180,E1 34914.123,E2 34914.123} C_VEL
LIN {X 0,Y 751.874,Z 167.503,A -85,B 0,C 180,E1 34911.896,E2 34911.896} C_VEL
LIN {X 0,Y 751.962,Z 167.504,A -85,B 0,C 180,E1 34909.194,E2 34909.194} C_VEL
LIN {X 0,Y 751.877,Z 167.503,A -85,B 0,C 180,E1 34906.408,E2 34906.408} C_VEL
LIN {X 0,Y 751.87,Z 167.504,A -85,B 0,C 180,E1 34904.179,E2 34904.179} C_VEL
LIN {X 0,Y 751.89,Z 167.503,A -85,B 0,C 180,E1 34901.789,E2 34901.789} C_VEL
LIN {X 0,Y 751.9,Z 167.503,A -85,B 0,C 180,E1 34898.76,E2 34898.76} C_VEL
LIN {X 0,Y 751.871,Z 167.504,A -85,B 0,C 180,E1 34896.37,E2 34896.37} C_VEL
LIN {X 0,Y 751.876,Z 167.503,A -85,B 0,C 180,E1 34894.054,E2 34894.054} C_VEL
LIN {X 0,Y 751.974,Z 167.501,A -85,B 0,C 180,E1 34891.313,E2 34891.313} C_VEL
LIN {X 0,Y 751.875,Z 167.504,A -85,B 0,C 180,E1 34888.58,E2 34888.58} C_VEL
LIN {X 0,Y 751.87,Z 167.503,A -85,B 0,C 180,E1 34886.32,E2 34886.32} C_VEL
LIN {X 0,Y 751.895,Z 167.503,A -85,B 0,C 180,E1 34883.942,E2 34883.942} C_VEL
LIN {X 0,Y 751.896,Z 167.503,A -85,B 0,C 180,E1 34880.925,E2 34880.925} C_VEL
LIN {X 0,Y 751.871,Z 167.504,A -85,B 0,C 180,E1 34878.526,E2 34878.526} C_VEL
LIN {X 0,Y 751.877,Z 167.503,A -85,B 0,C 180,E1 34876.249,E2 34876.249} C_VEL
LIN {X 0,Y 751.965,Z 167.503,A -85,B 0,C 180,E1 34873.446,E2 34873.446} C_VEL
LIN {X 0,Y 751.875,Z 167.504,A -85,B 0,C 180,E1 34870.759,E2 34870.759} C_VEL
LIN {X 0,Y 751.871,Z 167.502,A -85,B 0,C 180,E1 34868.484,E2 34868.484} C_VEL
LIN {X 0,Y 751.906,Z 167.503,A -85,B 0,C 180,E1 34866.048,E2 34866.048} C_VEL
LIN {X 0,Y 751.893,Z 167.501,A -85,B 0,C 180,E1 34863.092,E2 34863.092} C_VEL
LIN {X 0,Y 751.871,Z 167.505,A -85,B 0,C 180,E1 34860.704,E2 34860.704} C_VEL
LIN {X 0,Y 751.961,Z 167.825,A -85,B 0,C 180,E1 34860.054,E2 34860.054} C_VEL
LIN {X 0,Y 752.494,Z 170.743,A -85,B 0,C 180,E1 34859.794,E2 34859.794} C_VEL
LIN {X 0,Y 752.379,Z 207.1,A -85,B 0,C 180,E1 34857.029,E2 34857.029} C_VEL
LIN {X 0,Y 752.4,Z 226.446,A -85,B 0,C 180,E1 34855.606,E2 34855.606} C_VEL
LIN {X 0,Y 752.658,Z 232.103,A -85,B 0,C 180,E1 34855.529,E2 34855.529} C_VEL
LIN {X 0,Y 752.524,Z 505.253,A -85,B 0,C 180,E1 34852.736,E2 34852.736} C_VEL
LIN {X 0,Y 752.483,Z 534.401,A -85,B 0,C 180,E1 34852.396,E2 34852.396} C_VEL
LIN {X 0,Y 752.456,Z 556.195,A -85,B 0,C 180,E1 34852.001,E2 34852.001} C_VEL
LIN {X 0,Y 752.398,Z 576.494,A -85,B 0,C 180,E1 34851.494,E2 34851.494} C_VEL
LIN {X 0,Y 752.338,Z 596.755,A -85,B 0,C 180,E1 34850.863,E2 34850.863} C_VEL
LIN {X 0,Y 752.301,Z 617.781,A -85,B 0,C 180,E1 34850.051,E2 34850.051} C_VEL
LIN {X 0,Y 752.23,Z 636.759,A -85,B 0,C 180,E1 34849.164,E2 34849.164} C_VEL
LIN {X 0,Y 752.166,Z 655.166,A -85,B 0,C 180,E1 34848.161,E2 34848.161} C_VEL
LIN {X 0,Y 752.112,Z 673.281,A -85,B 0,C 180,E1 34847.004,E2 34847.004} C_VEL
LIN {X 0,Y 752.061,Z 690.237,A -85,B 0,C 180,E1 34845.735,E2 34845.735} C_VEL
LIN {X 0,Y 752.013,Z 705.586,A -85,B 0,C 180,E1 34844.395,E2 34844.395} C_VEL
LIN {X 0,Y 751.975,Z 719.46,A -85,B 0,C 180,E1 34842.984,E2 34842.984} C_VEL
LIN {X 0,Y 751.952,Z 731.356,A -85,B 0,C 180,E1 34841.581,E2 34841.581} C_VEL
LIN {X 0,Y 751.94,Z 742.37,A -85,B 0,C 180,E1 34840.031,E2 34840.031} C_VEL
LIN {X 0,Y 751.912,Z 751.479,A -85,B 0,C 180,E1 34838.487,E2 34838.487} C_VEL
LIN {X 0,Y 751.911,Z 758.93,A -85,B 0,C 180,E1 34836.95,E2 34836.95} C_VEL
LIN {X 0,Y 751.915,Z 764.909,A -85,B 0,C 180,E1 34835.34,E2 34835.34} C_VEL
LIN {X 0,Y 751.915,Z 769.625,A -85,B 0,C 180,E1 34833.583,E2 34833.583} C_VEL
LIN {X 0,Y 751.919,Z 772.418,A -85,B 0,C 180,E1 34831.905,E2 34831.905} C_VEL
LIN {X 0,Y 751.903,Z 773.44,A -85,B 0,C 180,E1 34830.229,E2 34830.229} C_VEL
LIN {X 0,Y 751.898,Z 772.818,A -85,B 0,C 180,E1 34828.552,E2 34828.552} C_VEL
LIN {X 0,Y 751.897,Z 770.571,A -85,B 0,C 180,E1 34826.875,E2 34826.875} C_VEL
LIN {X 0,Y 751.904,Z 766.987,A -85,B 0,C 180,E1 34825.348,E2 34825.348} C_VEL
LIN {X 0,Y 751.917,Z 761.375,A -85,B 0,C 180,E1 34823.664,E2 34823.664} C_VEL
LIN {X 0,Y 751.93,Z 754.314,A -85,B 0,C 180,E1 34822.052,E2 34822.052} C_VEL
LIN {X 0,Y 751.925,Z 745.754,A -85,B 0,C 180,E1 34820.51,E2 34820.51} C_VEL
LIN {X 0,Y 751.944,Z 735.077,A -85,B 0,C 180,E1 34818.918,E2 34818.918} C_VEL
LIN {X 0,Y 751.972,Z 722.986,A -85,B 0,C 180,E1 34817.406,E2 34817.406} C_VEL
LIN {X 0,Y 752.005,Z 709.695,A -85,B 0,C 180,E1 34815.998,E2 34815.998} C_VEL
LIN {X 0,Y 752.044,Z 694.976,A -85,B 0,C 180,E1 34814.66,E2 34814.66} C_VEL
LIN {X 0,Y 752.097,Z 678.259,A -85,B 0,C 180,E1 34813.354,E2 34813.354} C_VEL
LIN {X 0,Y 752.159,Z 661.114,A -85,B 0,C 180,E1 34812.199,E2 34812.199} C_VEL
LIN {X 0,Y 752.216,Z 642.333,A -85,B 0,C 180,E1 34811.117,E2 34811.117} C_VEL
LIN {X 0,Y 752.273,Z 623.226,A -85,B 0,C 180,E1 34810.191,E2 34810.191} C_VEL
LIN {X 0,Y 752.333,Z 602.194,A -85,B 0,C 180,E1 34809.335,E2 34809.335} C_VEL
LIN {X 0,Y 752.397,Z 581.637,A -85,B 0,C 180,E1 34808.649,E2 34808.649} C_VEL
LIN {X 0,Y 752.441,Z 560.279,A -85,B 0,C 180,E1 34808.092,E2 34808.092} C_VEL
LIN {X 0,Y 752.479,Z 538.254,A -85,B 0,C 180,E1 34807.665,E2 34807.665} C_VEL
LIN {X 0,Y 752.512,Z 515.301,A -85,B 0,C 180,E1 34807.366,E2 34807.366} C_VEL
LIN {X 0,Y 752.653,Z 244.939,A -85,B 0,C 180,E1 34804.604,E2 34804.604} C_VEL
LIN {X 0,Y 752.514,Z 227.114,A -85,B 0,C 180,E1 34804.411,E2 34804.411} C_VEL
LIN {X 0,Y 752.338,Z 224.928,A -85,B 0,C 180,E1 34804.303,E2 34804.303} C_VEL
LIN {X 0,Y 752.447,Z 187.785,A -85,B 0,C 180,E1 34801.511,E2 34801.511} C_VEL
LIN {X 0,Y 752.283,Z 169.062,A -85,B 0,C 180,E1 34800.066,E2 34800.066} C_VEL
LIN {X 0,Y 751.92,Z 167.605,A -85,B 0,C 180,E1 34799.895,E2 34799.895} C_VEL
LIN {X 0,Y 751.871,Z 167.502,A -85,B 0,C 180,E1 34797.417,E2 34797.417} C_VEL
LIN {X 0,Y 751.884,Z 167.504,A -85,B 0,C 180,E1 34795.034,E2 34795.034} C_VEL
LIN {X 0,Y 751.936,Z 167.502,A -85,B 0,C 180,E1 34792.174,E2 34792.174} C_VEL
LIN {X 0,Y 751.875,Z 167.504,A -85,B 0,C 180,E1 34789.642,E2 34789.642} C_VEL
LIN {X 0,Y 751.87,Z 167.503,A -85,B 0,C 180,E1 34787.405,E2 34787.405} C_VEL
LIN {X 0,Y 751.888,Z 167.504,A -85,B 0,C 180,E1 34785.086,E2 34785.086} C_VEL
LIN {X 0,Y 751.908,Z 167.504,A -85,B 0,C 180,E1 34782.104,E2 34782.104} C_VEL
LIN {X 0,Y 751.871,Z 167.503,A -85,B 0,C 180,E1 34779.656,E2 34779.656} C_VEL
LIN {X 0,Y 751.878,Z 167.504,A -85,B 0,C 180,E1 34777.331,E2 34777.331} C_VEL
LIN {X 0,Y 751.973,Z 167.503,A -85,B 0,C 180,E1 34774.596,E2 34774.596} C_VEL
LIN {X 0,Y 751.874,Z 167.504,A -85,B 0,C 180,E1 34771.825,E2 34771.825} C_VEL
LIN {X 0,Y 751.871,Z 167.502,A -85,B 0,C 180,E1 34769.563,E2 34769.563} C_VEL
LIN {X 0,Y 751.904,Z 167.501,A -85,B 0,C 180,E1 34767.138,E2 34767.138} C_VEL
LIN {X 0,Y 751.893,Z 167.504,A -85,B 0,C 180,E1 34764.179,E2 34764.179} C_VEL
LIN {X 0,Y 751.87,Z 167.503,A -85,B 0,C 180,E1 34761.78,E2 34761.78} C_VEL
LIN {X 0,Y 751.879,Z 167.504,A -85,B 0,C 180,E1 34759.483,E2 34759.483} C_VEL
LIN {X 0,Y 751.958,Z 167.504,A -85,B 0,C 180,E1 34756.692,E2 34756.692} C_VEL
LIN {X 0,Y 751.877,Z 167.503,A -85,B 0,C 180,E1 34754.085,E2 34754.085} C_VEL
LIN {X 0,Y 751.87,Z 167.503,A -85,B 0,C 180,E1 34751.818,E2 34751.818} C_VEL
LIN {X 0,Y 751.904,Z 167.503,A -85,B 0,C 180,E1 34749.337,E2 34749.337} C_VEL
LIN {X 0,Y 751.889,Z 167.504,A -85,B 0,C 180,E1 34746.337,E2 34746.337} C_VEL
LIN {X 0,Y 751.87,Z 167.503,A -85,B 0,C 180,E1 34744.042,E2 34744.042} C_VEL
LIN {X 0,Y 751.875,Z 167.503,A -85,B 0,C 180,E1 34741.753,E2 34741.753} C_VEL
LIN {X 0,Y 751.977,Z 167.504,A -85,B 0,C 180,E1 34739.01,E2 34739.01} C_VEL
LIN {X 0,Y 751.874,Z 167.504,A -85,B 0,C 180,E1 34736.264,E2 34736.264} C_VEL
LIN {X 0,Y 751.875,Z 167.504,A -85,B 0,C 180,E1 34734.304,E2 34734.304} C_VEL
LIN {X 0,Y 750.861,Z 167.633,A -85,B 0,C 180,E1 34733.717,E2 34733.717} C_VEL
LIN {X 0,Y 744.449,Z 168.429,A -85,B 0,C 180,E1 34732.073,E2 34732.073} C_VEL
LIN {X 0,Y 743.952,Z 168.492,A -85,B 0,C 180,E1 34731.646,E2 34731.646} C_VEL
LIN {X 0,Y 743.957,Z 168.492,A -85,B 0,C 180,E1 34728.605,E2 34728.605} C_VEL
LIN {X 0,Y 743.93,Z 168.493,A -85,B 0,C 180,E1 34726.158,E2 34726.158} C_VEL
LIN {X 0,Y 743.942,Z 168.492,A -85,B 0,C 180,E1 34723.846,E2 34723.846} C_VEL
LIN {X 0,Y 744.004,Z 168.493,A -85,B 0,C 180,E1 34721.02,E2 34721.02} C_VEL
LIN {X 0,Y 743.933,Z 168.492,A -85,B 0,C 180,E1 34718.391,E2 34718.391} C_VEL
LIN {X 0,Y 743.936,Z 168.493,A -85,B 0,C 180,E1 34716.04,E2 34716.04} C_VEL
LIN {X 0,Y 744.025,Z 168.488,A -85,B 0,C 180,E1 34713.243,E2 34713.243} C_VEL
LIN {X 0,Y 743.935,Z 168.492,A -85,B 0,C 180,E1 34710.533,E2 34710.533} C_VEL
LIN {X 0,Y 743.931,Z 168.493,A -85,B 0,C 180,E1 34708.285,E2 34708.285} C_VEL
LIN {X 0,Y 743.976,Z 168.492,A -85,B 0,C 180,E1 34705.727,E2 34705.727} C_VEL
LIN {X 0,Y 743.945,Z 168.493,A -85,B 0,C 180,E1 34702.784,E2 34702.784} C_VEL
LIN {X 0,Y 743.93,Z 168.493,A -85,B 0,C 180,E1 34700.425,E2 34700.425} C_VEL
LIN {X 0,Y 743.946,Z 168.493,A -85,B 0,C 180,E1 34698.088,E2 34698.088} C_VEL
LIN {X 0,Y 743.984,Z 168.493,A -85,B 0,C 180,E1 34695.196,E2 34695.196} C_VEL
LIN {X 0,Y 743.931,Z 168.493,A -85,B 0,C 180,E1 34692.634,E2 34692.634} C_VEL
LIN {X 0,Y 743.934,Z 168.493,A -85,B 0,C 180,E1 34690.352,E2 34690.352} C_VEL
LIN {X 0,Y 744.033,Z 168.493,A -85,B 0,C 180,E1 34687.592,E2 34687.592} C_VEL
LIN {X 0,Y 743.934,Z 168.493,A -85,B 0,C 180,E1 34684.793,E2 34684.793} C_VEL
LIN {X 0,Y 743.935,Z 168.493,A -85,B 0,C 180,E1 34682.426,E2 34682.426} C_VEL
LIN {X 0,Y 744.033,Z 168.493,A -85,B 0,C 180,E1 34679.635,E2 34679.635} C_VEL
LIN {X 0,Y 743.932,Z 168.493,A -85,B 0,C 180,E1 34676.843,E2 34676.843} C_VEL
LIN {X 0,Y 743.935,Z 168.493,A -85,B 0,C 180,E1 34674.504,E2 34674.504} C_VEL
LIN {X 0,Y 744.032,Z 168.493,A -85,B 0,C 180,E1 34671.769,E2 34671.769} C_VEL
LIN {X 0,Y 743.938,Z 168.494,A -85,B 0,C 180,E1 34669.06,E2 34669.06} C_VEL
LIN {X 0,Y 743.931,Z 168.493,A -85,B 0,C 180,E1 34666.714,E2 34666.714} C_VEL
LIN {X 0,Y 743.982,Z 168.494,A -85,B 0,C 180,E1 34664.156,E2 34664.156} C_VEL
LIN {X 0,Y 743.944,Z 168.494,A -85,B 0,C 180,E1 34661.236,E2 34661.236} C_VEL
LIN {X 0,Y 743.929,Z 168.493,A -85,B 0,C 180,E1 34658.89,E2 34658.89} C_VEL
LIN {X 0,Y 743.944,Z 168.494,A -85,B 0,C 180,E1 34656.559,E2 34656.559} C_VEL
LIN {X 0,Y 743.976,Z 168.494,A -85,B 0,C 180,E1 34653.621,E2 34653.621} C_VEL
LIN {X 0,Y 743.933,Z 168.494,A -85,B 0,C 180,E1 34651.155,E2 34651.155} C_VEL
LIN {X 0,Y 743.929,Z 168.494,A -85,B 0,C 180,E1 34648.922,E2 34648.922} C_VEL
LIN {X 0,Y 743.966,Z 168.494,A -85,B 0,C 180,E1 34646.456,E2 34646.456} C_VEL
LIN {X 0,Y 743.952,Z 168.494,A -85,B 0,C 180,E1 34643.518,E2 34643.518} C_VEL
LIN {X 0,Y 743.93,Z 168.493,A -85,B 0,C 180,E1 34641.187,E2 34641.187} C_VEL
LIN {X 0,Y 743.938,Z 168.494,A -85,B 0,C 180,E1 34638.842,E2 34638.842} C_VEL
LIN {X 0,Y 744.009,Z 168.494,A -85,B 0,C 180,E1 34636.003,E2 34636.003} C_VEL
LIN {X 0,Y 743.933,Z 168.493,A -85,B 0,C 180,E1 34633.367,E2 34633.367} C_VEL
LIN {X 0,Y 743.934,Z 168.493,A -85,B 0,C 180,E1 34631.021,E2 34631.021} C_VEL
LIN {X 0,Y 744.021,Z 168.494,A -85,B 0,C 180,E1 34628.314,E2 34628.314} C_VEL
LIN {X 0,Y 743.939,Z 168.493,A -85,B 0,C 180,E1 34625.549,E2 34625.549} C_VEL
LIN {X 0,Y 743.93,Z 168.493,A -85,B 0,C 180,E1 34623.244,E2 34623.244} C_VEL
LIN {X 0,Y 743.971,Z 168.493,A -85,B 0,C 180,E1 34620.716,E2 34620.716} C_VEL
LIN {X 0,Y 743.947,Z 168.493,A -85,B 0,C 180,E1 34617.757,E2 34617.757} C_VEL
LIN {X 0,Y 743.93,Z 168.493,A -85,B 0,C 180,E1 34615.343,E2 34615.343} C_VEL
LIN {X 0,Y 743.974,Z 168.493,A -85,B 0,C 180,E1 34612.792,E2 34612.792} C_VEL
LIN {X 0,Y 743.946,Z 168.493,A -85,B 0,C 180,E1 34609.831,E2 34609.831} C_VEL
LIN {X 0,Y 743.931,Z 168.493,A -85,B 0,C 180,E1 34607.552,E2 34607.552} C_VEL
LIN {X 0,Y 743.939,Z 168.493,A -85,B 0,C 180,E1 34605.207,E2 34605.207} C_VEL
LIN {X 0,Y 744.016,Z 168.493,A -85,B 0,C 180,E1 34602.427,E2 34602.427} C_VEL
LIN {X 0,Y 743.935,Z 168.493,A -85,B 0,C 180,E1 34599.763,E2 34599.763} C_VEL
LIN {X 0,Y 743.933,Z 168.493,A -85,B 0,C 180,E1 34597.41,E2 34597.41} C_VEL
LIN {X 0,Y 744.03,Z 168.489,A -85,B 0,C 180,E1 34594.643,E2 34594.643} C_VEL
LIN {X 0,Y 743.935,Z 168.493,A -85,B 0,C 180,E1 34591.862,E2 34591.862} C_VEL
LIN {X 0,Y 743.932,Z 168.492,A -85,B 0,C 180,E1 34589.556,E2 34589.556} C_VEL
LIN {X 0,Y 743.97,Z 168.487,A -85,B 0,C 180,E1 34587.105,E2 34587.105} C_VEL
LIN {X 0,Y 743.947,Z 168.493,A -85,B 0,C 180,E1 34584.116,E2 34584.116} C_VEL
LIN {X 0,Y 743.93,Z 168.492,A -85,B 0,C 180,E1 34581.775,E2 34581.775} C_VEL
LIN {X 0,Y 743.949,Z 168.493,A -85,B 0,C 180,E1 34579.389,E2 34579.389} C_VEL
LIN {X 0,Y 743.966,Z 168.492,A -85,B 0,C 180,E1 34576.394,E2 34576.394} C_VEL
LIN {X 0,Y 743.932,Z 168.493,A -85,B 0,C 180,E1 34574.001,E2 34574.001} C_VEL
LIN {X 0,Y 743.937,Z 168.491,A -85,B 0,C 180,E1 34571.631,E2 34571.631} C_VEL
LIN {X 0,Y 744.02,Z 168.492,A -85,B 0,C 180,E1 34568.813,E2 34568.813} C_VEL
LIN {X 0,Y 743.936,Z 168.492,A -85,B 0,C 180,E1 34566.173,E2 34566.173} C_VEL
LIN {X 0,Y 743.931,Z 168.493,A -85,B 0,C 180,E1 34563.853,E2 34563.853} C_VEL
LIN {X 0,Y 743.981,Z 168.491,A -85,B 0,C 180,E1 34561.309,E2 34561.309} C_VEL
LIN {X 0,Y 743.945,Z 168.492,A -85,B 0,C 180,E1 34558.383,E2 34558.383} C_VEL
LIN {X 0,Y 743.931,Z 168.492,A -85,B 0,C 180,E1 34556.069,E2 34556.069} C_VEL
LIN {X 0,Y 743.943,Z 168.493,A -85,B 0,C 180,E1 34553.75,E2 34553.75} C_VEL
LIN {X 0,Y 744.01,Z 168.492,A -85,B 0,C 180,E1 34550.953,E2 34550.953} C_VEL
LIN {X 0,Y 743.934,Z 168.492,A -85,B 0,C 180,E1 34548.29,E2 34548.29} C_VEL
LIN {X 0,Y 743.938,Z 168.492,A -85,B 0,C 180,E1 34545.92,E2 34545.92} C_VEL
LIN {X 0,Y 744.026,Z 168.493,A -85,B 0,C 180,E1 34543.206,E2 34543.206} C_VEL
LIN {X 0,Y 743.936,Z 168.493,A -85,B 0,C 180,E1 34540.447,E2 34540.447} C_VEL
LIN {X 0,Y 743.933,Z 168.492,A -85,B 0,C 180,E1 34538.142,E2 34538.142} C_VEL
LIN {X 0,Y 744.006,Z 168.493,A -85,B 0,C 180,E1 34535.463,E2 34535.463} C_VEL
LIN {X 0,Y 743.942,Z 168.489,A -85,B 0,C 180,E1 34532.634,E2 34532.634} C_VEL
LIN {X 0,Y 743.932,Z 168.491,A -85,B 0,C 180,E1 34530.355,E2 34530.355} C_VEL
LIN {X 0,Y 743.945,Z 168.493,A -85,B 0,C 180,E1 34528.025,E2 34528.025} C_VEL
LIN {X 0,Y 743.997,Z 168.491,A -85,B 0,C 180,E1 34525.167,E2 34525.167} C_VEL
LIN {X 0,Y 743.934,Z 168.493,A -85,B 0,C 180,E1 34522.582,E2 34522.582} C_VEL
LIN {X 0,Y 743.938,Z 168.491,A -85,B 0,C 180,E1 34520.225,E2 34520.225} C_VEL
LIN {X 0,Y 744.03,Z 168.492,A -85,B 0,C 180,E1 34517.421,E2 34517.421} C_VEL
LIN {X 0,Y 743.935,Z 168.493,A -85,B 0,C 180,E1 34514.683,E2 34514.683} C_VEL
LIN {X 0,Y 743.936,Z 168.492,A -85,B 0,C 180,E1 34512.334,E2 34512.334} C_VEL
LIN {X 0,Y 744.024,Z 168.494,A -85,B 0,C 180,E1 34509.641,E2 34509.641} C_VEL
LIN {X 0,Y 743.941,Z 168.491,A -85,B 0,C 180,E1 34506.897,E2 34506.897} C_VEL
LIN {X 0,Y 743.933,Z 168.493,A -85,B 0,C 180,E1 34504.522,E2 34504.522} C_VEL
LIN {X 0,Y 743.999,Z 168.489,A -85,B 0,C 180,E1 34501.877,E2 34501.877} C_VEL
LIN {X 0,Y 743.984,Z 168.771,A -85,B 0,C 180,E1 34500.337,E2 34500.337} C_VEL
LIN {X 0,Y 745.074,Z 173.015,A -85,B 0,C 180,E1 34499.944,E2 34499.944} C_VEL
LIN {X 0,Y 744.857,Z 209.373,A -85,B 0,C 180,E1 34497.152,E2 34497.152} C_VEL
LIN {X 0,Y 744.846,Z 226.425,A -85,B 0,C 180,E1 34495.885,E2 34495.885} C_VEL
LIN {X 0,Y 745.436,Z 230.797,A -85,B 0,C 180,E1 34495.808,E2 34495.808} C_VEL
LIN {X 0,Y 745.142,Z 503.917,A -85,B 0,C 180,E1 34492.987,E2 34492.987} C_VEL
LIN {X 0,Y 745.073,Z 533.877,A -85,B 0,C 180,E1 34492.64,E2 34492.64} C_VEL
LIN {X 0,Y 745.01,Z 555.999,A -85,B 0,C 180,E1 34492.236,E2 34492.236} C_VEL
LIN {X 0,Y 744.901,Z 576.415,A -85,B 0,C 180,E1 34491.723,E2 34491.723} C_VEL
LIN {X 0,Y 744.789,Z 596.773,A -85,B 0,C 180,E1 34491.084,E2 34491.084} C_VEL
LIN {X 0,Y 744.692,Z 617.78,A -85,B 0,C 180,E1 34490.265,E2 34490.265} C_VEL
LIN {X 0,Y 744.553,Z 636.754,A -85,B 0,C 180,E1 34489.37,E2 34489.37} C_VEL
LIN {X 0,Y 744.426,Z 655.173,A -85,B 0,C 180,E1 34488.357,E2 34488.357} C_VEL
LIN {X 0,Y 744.321,Z 673.273,A -85,B 0,C 180,E1 34487.187,E2 34487.187} C_VEL
LIN {X 0,Y 744.22,Z 689.732,A -85,B 0,C 180,E1 34485.945,E2 34485.945} C_VEL
LIN {X 0,Y 744.125,Z 704.742,A -85,B 0,C 180,E1 34484.63,E2 34484.63} C_VEL
LIN {X 0,Y 744.043,Z 719.459,A -85,B 0,C 180,E1 34483.125,E2 34483.125} C_VEL
LIN {X 0,Y 744,Z 731.348,A -85,B 0,C 180,E1 34481.707,E2 34481.707} C_VEL
LIN {X 0,Y 743.964,Z 742.373,A -85,B 0,C 180,E1 34480.139,E2 34480.139} C_VEL
LIN {X 0,Y 743.927,Z 751.48,A -85,B 0,C 180,E1 34478.579,E2 34478.579} C_VEL
LIN {X 0,Y 743.923,Z 758.924,A -85,B 0,C 180,E1 34477.025,E2 34477.025} C_VEL
LIN {X 0,Y 743.918,Z 764.911,A -85,B 0,C 180,E1 34475.398,E2 34475.398} C_VEL
LIN {X 0,Y 743.916,Z 769.626,A -85,B 0,C 180,E1 34473.621,E2 34473.621} C_VEL
LIN {X 0,Y 743.919,Z 772.413,A -85,B 0,C 180,E1 34471.925,E2 34471.925} C_VEL
LIN {X 0,Y 743.903,Z 773.44,A -85,B 0,C 180,E1 34470.231,E2 34470.231} C_VEL
LIN {X 0,Y 743.899,Z 772.821,A -85,B 0,C 180,E1 34468.537,E2 34468.537} C_VEL
LIN {X 0,Y 743.897,Z 770.572,A -85,B 0,C 180,E1 34466.841,E2 34466.841} C_VEL
LIN {X 0,Y 743.902,Z 766.985,A -85,B 0,C 180,E1 34465.298,E2 34465.298} C_VEL
LIN {X 0,Y 743.917,Z 761.379,A -85,B 0,C 180,E1 34463.596,E2 34463.596} C_VEL
LIN {X 0,Y 743.936,Z 754.308,A -85,B 0,C 180,E1 34461.966,E2 34461.966} C_VEL
LIN {X 0,Y 743.949,Z 745.753,A -85,B 0,C 180,E1 34460.408,E2 34460.408} C_VEL
LIN {X 0,Y 743.989,Z 734.832,A -85,B 0,C 180,E1 34458.764,E2 34458.764} C_VEL
LIN {X 0,Y 744.041,Z 722.98,A -85,B 0,C 180,E1 34457.27,E2 34457.27} C_VEL
LIN {X 0,Y 744.102,Z 709.693,A -85,B 0,C 180,E1 34455.846,E2 34455.846} C_VEL
LIN {X 0,Y 744.182,Z 694.981,A -85,B 0,C 180,E1 34454.494,E2 34454.494} C_VEL
LIN {X 0,Y 744.282,Z 678.122,A -85,B 0,C 180,E1 34453.164,E2 34453.164} C_VEL
LIN {X 0,Y 744.408,Z 660.805,A -85,B 0,C 180,E1 34451.988,E2 34451.988} C_VEL
LIN {X 0,Y 744.538,Z 641.568,A -85,B 0,C 180,E1 34450.874,E2 34450.874} C_VEL
LIN {X 0,Y 744.644,Z 622.34,A -85,B 0,C 180,E1 34449.938,E2 34449.938} C_VEL
LIN {X 0,Y 744.767,Z 602.365,A -85,B 0,C 180,E1 34449.121,E2 34449.121} C_VEL
LIN {X 0,Y 744.894,Z 580.897,A -85,B 0,C 180,E1 34448.403,E2 34448.403} C_VEL
LIN {X 0,Y 744.983,Z 559.859,A -85,B 0,C 180,E1 34447.851,E2 34447.851} C_VEL
LIN {X 0,Y 745.066,Z 537.97,A -85,B 0,C 180,E1 34447.425,E2 34447.425} C_VEL
LIN {X 0,Y 745.128,Z 513.775,A -85,B 0,C 180,E1 34447.113,E2 34447.113} C_VEL
LIN {X 0,Y 745.423,Z 243.424,A -85,B 0,C 180,E1 34444.324,E2 34444.324} C_VEL
LIN {X 0,Y 745.218,Z 228.245,A -85,B 0,C 180,E1 34444.157,E2 34444.157} C_VEL
LIN {X 0,Y 744.81,Z 225.896,A -85,B 0,C 180,E1 34444.088,E2 34444.088} C_VEL
LIN {X 0,Y 744.984,Z 188.921,A -85,B 0,C 180,E1 34441.287,E2 34441.287} C_VEL
LIN {X 0,Y 744.893,Z 171.878,A -85,B 0,C 180,E1 34439.959,E2 34439.959} C_VEL
LIN {X 0,Y 743.963,Z 168.641,A -85,B 0,C 180,E1 34439.639,E2 34439.639} C_VEL
LIN {X 0,Y 743.933,Z 168.489,A -85,B 0,C 180,E1 34437.287,E2 34437.287} C_VEL
LIN {X 0,Y 743.984,Z 168.493,A -85,B 0,C 180,E1 34434.702,E2 34434.702} C_VEL
LIN {X 0,Y 743.95,Z 168.49,A -85,B 0,C 180,E1 34431.818,E2 34431.818} C_VEL
LIN {X 0,Y 743.933,Z 168.494,A -85,B 0,C 180,E1 34429.527,E2 34429.527} C_VEL
LIN {X 0,Y 743.937,Z 168.492,A -85,B 0,C 180,E1 34427.262,E2 34427.262} C_VEL
LIN {X 0,Y 744.032,Z 168.491,A -85,B 0,C 180,E1 34424.479,E2 34424.479} C_VEL
LIN {X 0,Y 743.938,Z 168.493,A -85,B 0,C 180,E1 34421.768,E2 34421.768} C_VEL
LIN {X 0,Y 743.933,Z 168.491,A -85,B 0,C 180,E1 34419.475,E2 34419.475} C_VEL
LIN {X 0,Y 743.981,Z 168.493,A -85,B 0,C 180,E1 34416.912,E2 34416.912} C_VEL
LIN {X 0,Y 743.948,Z 168.492,A -85,B 0,C 180,E1 34413.988,E2 34413.988} C_VEL
LIN {X 0,Y 743.931,Z 168.493,A -85,B 0,C 180,E1 34411.614,E2 34411.614} C_VEL
LIN {X 0,Y 743.947,Z 168.491,A -85,B 0,C 180,E1 34409.29,E2 34409.29} C_VEL
LIN {X 0,Y 743.975,Z 168.492,A -85,B 0,C 180,E1 34406.329,E2 34406.329} C_VEL
LIN {X 0,Y 743.932,Z 168.493,A -85,B 0,C 180,E1 34403.78,E2 34403.78} C_VEL
LIN {X 0,Y 743.942,Z 168.491,A -85,B 0,C 180,E1 34401.443,E2 34401.443} C_VEL
LIN {X 0,Y 744.015,Z 168.491,A -85,B 0,C 180,E1 34398.654,E2 34398.654} C_VEL
LIN {X 0,Y 743.935,Z 168.493,A -85,B 0,C 180,E1 34395.994,E2 34395.994} C_VEL
LIN {X 0,Y 743.932,Z 168.492,A -85,B 0,C 180,E1 34393.763,E2 34393.763} C_VEL
LIN {X 0,Y 743.975,Z 168.492,A -85,B 0,C 180,E1 34391.238,E2 34391.238} C_VEL
LIN {X 0,Y 743.954,Z 168.491,A -85,B 0,C 180,E1 34388.346,E2 34388.346} C_VEL
LIN {X 0,Y 743.933,Z 168.493,A -85,B 0,C 180,E1 34386.018,E2 34386.018} C_VEL
LIN {X 0,Y 743.938,Z 168.492,A -85,B 0,C 180,E1 34383.699,E2 34383.699} C_VEL
LIN {X 0,Y 744.028,Z 168.493,A -85,B 0,C 180,E1 34380.924,E2 34380.924} C_VEL
LIN {X 0,Y 743.935,Z 168.491,A -85,B 0,C 180,E1 34378.229,E2 34378.229} C_VEL
LIN {X 0,Y 743.931,Z 168.493,A -85,B 0,C 180,E1 34375.915,E2 34375.915} C_VEL
LIN {X 0,Y 743.999,Z 168.492,A -85,B 0,C 180,E1 34373.285,E2 34373.285} C_VEL
LIN {X 0,Y 743.952,Z 168.492,A -85,B 0,C 180,E1 34371.646,E2 34371.646} C_VEL
LIN {X 0,Y 743.023,Z 168.619,A -85,B 0,C 180,E1 34371.053,E2 34371.053} C_VEL
LIN {X 0,Y 736.546,Z 169.428,A -85,B 0,C 180,E1 34369.349,E2 34369.349} C_VEL
LIN {X 0,Y 736.07,Z 169.48,A -85,B 0,C 180,E1 34368.96,E2 34368.96} C_VEL
LIN {X 0,Y 735.995,Z 169.482,A -85,B 0,C 180,E1 34366.326,E2 34366.326} C_VEL
LIN {X 0,Y 735.992,Z 169.481,A -85,B 0,C 180,E1 34364.072,E2 34364.072} C_VEL
LIN {X 0,Y 736.053,Z 169.481,A -85,B 0,C 180,E1 34361.454,E2 34361.454} C_VEL
LIN {X 0,Y 736.005,Z 169.48,A -85,B 0,C 180,E1 34358.565,E2 34358.565} C_VEL
LIN {X 0,Y 735.993,Z 169.482,A -85,B 0,C 180,E1 34356.203,E2 34356.203} C_VEL
LIN {X 0,Y 736.04,Z 169.48,A -85,B 0,C 180,E1 34353.626,E2 34353.626} C_VEL
LIN {X 0,Y 736.007,Z 169.48,A -85,B 0,C 180,E1 34350.699,E2 34350.699} C_VEL
LIN {X 0,Y 735.992,Z 169.482,A -85,B 0,C 180,E1 34348.372,E2 34348.372} C_VEL
LIN {X 0,Y 736.02,Z 169.48,A -85,B 0,C 180,E1 34345.87,E2 34345.87} C_VEL
LIN {X 0,Y 736.015,Z 169.482,A -85,B 0,C 180,E1 34342.877,E2 34342.877} C_VEL
LIN {X 0,Y 735.992,Z 169.482,A -85,B 0,C 180,E1 34340.494,E2 34340.494} C_VEL
LIN {X 0,Y 736.001,Z 169.482,A -85,B 0,C 180,E1 34338.16,E2 34338.16} C_VEL
LIN {X 0,Y 736.077,Z 169.482,A -85,B 0,C 180,E1 34335.374,E2 34335.374} C_VEL
LIN {X 0,Y 735.994,Z 169.482,A -85,B 0,C 180,E1 34332.674,E2 34332.674} C_VEL
LIN {X 0,Y 735.995,Z 169.482,A -85,B 0,C 180,E1 34330.387,E2 34330.387} C_VEL
LIN {X 0,Y 736.089,Z 169.482,A -85,B 0,C 180,E1 34327.633,E2 34327.633} C_VEL
LIN {X 0,Y 735.995,Z 169.482,A -85,B 0,C 180,E1 34324.786,E2 34324.786} C_VEL
LIN {X 0,Y 735.995,Z 169.482,A -85,B 0,C 180,E1 34322.449,E2 34322.449} C_VEL
LIN {X 0,Y 736.092,Z 169.482,A -85,B 0,C 180,E1 34319.629,E2 34319.629} C_VEL
LIN {X 0,Y 735.996,Z 169.482,A -85,B 0,C 180,E1 34316.894,E2 34316.894} C_VEL
LIN {X 0,Y 735.995,Z 169.483,A -85,B 0,C 180,E1 34314.561,E2 34314.561} C_VEL
LIN {X 0,Y 736.093,Z 169.482,A -85,B 0,C 180,E1 34311.764,E2 34311.764} C_VEL
LIN {X 0,Y 735.997,Z 169.483,A -85,B 0,C 180,E1 34308.993,E2 34308.993} C_VEL
LIN {X 0,Y 735.995,Z 169.482,A -85,B 0,C 180,E1 34306.655,E2 34306.655} C_VEL
LIN {X 0,Y 736.083,Z 169.483,A -85,B 0,C 180,E1 34303.91,E2 34303.91} C_VEL
LIN {X 0,Y 735.998,Z 169.483,A -85,B 0,C 180,E1 34301.121,E2 34301.121} C_VEL
LIN {X 0,Y 735.994,Z 169.483,A -85,B 0,C 180,E1 34298.751,E2 34298.751} C_VEL
LIN {X 0,Y 736.085,Z 169.483,A -85,B 0,C 180,E1 34296.003,E2 34296.003} C_VEL
LIN {X 0,Y 735.996,Z 169.483,A -85,B 0,C 180,E1 34293.193,E2 34293.193} C_VEL
LIN {X 0,Y 735.993,Z 169.483,A -85,B 0,C 180,E1 34290.856,E2 34290.856} C_VEL
LIN {X 0,Y 736.037,Z 169.483,A -85,B 0,C 180,E1 34288.365,E2 34288.365} C_VEL
LIN {X 0,Y 736.004,Z 169.483,A -85,B 0,C 180,E1 34285.403,E2 34285.403} C_VEL
LIN {X 0,Y 735.991,Z 169.483,A -85,B 0,C 180,E1 34283.056,E2 34283.056} C_VEL
LIN {X 0,Y 736.017,Z 169.483,A -85,B 0,C 180,E1 34280.619,E2 34280.619} C_VEL
LIN {X 0,Y 736.015,Z 169.482,A -85,B 0,C 180,E1 34277.607,E2 34277.607} C_VEL
LIN {X 0,Y 735.991,Z 169.483,A -85,B 0,C 180,E1 34275.204,E2 34275.204} C_VEL
LIN {X 0,Y 736.004,Z 169.482,A -85,B 0,C 180,E1 34272.857,E2 34272.857} C_VEL
LIN {X 0,Y 736.055,Z 169.483,A -85,B 0,C 180,E1 34269.984,E2 34269.984} C_VEL
LIN {X 0,Y 735.995,Z 169.482,A -85,B 0,C 180,E1 34267.392,E2 34267.392} C_VEL
LIN {X 0,Y 735.995,Z 169.483,A -85,B 0,C 180,E1 34265.096,E2 34265.096} C_VEL
LIN {X 0,Y 736.084,Z 169.483,A -85,B 0,C 180,E1 34262.322,E2 34262.322} C_VEL
LIN {X 0,Y 735.996,Z 169.482,A -85,B 0,C 180,E1 34259.558,E2 34259.558} C_VEL
LIN {X 0,Y 735.996,Z 169.482,A -85,B 0,C 180,E1 34257.181,E2 34257.181} C_VEL
LIN {X 0,Y 736.082,Z 169.483,A -85,B 0,C 180,E1 34254.361,E2 34254.361} C_VEL
LIN {X 0,Y 735.995,Z 169.482,A -85,B 0,C 180,E1 34251.618,E2 34251.618} C_VEL
LIN {X 0,Y 735.995,Z 169.482,A -85,B 0,C 180,E1 34249.295,E2 34249.295} C_VEL
LIN {X 0,Y 736.079,Z 169.483,A -85,B 0,C 180,E1 34246.587,E2 34246.587} C_VEL
LIN {X 0,Y 735.998,Z 169.482,A -85,B 0,C 180,E1 34243.749,E2 34243.749} C_VEL
LIN {X 0,Y 735.993,Z 169.482,A -85,B 0,C 180,E1 34241.424,E2 34241.424} C_VEL
LIN {X 0,Y 736.062,Z 169.482,A -85,B 0,C 180,E1 34238.773,E2 34238.773} C_VEL
LIN {X 0,Y 736.002,Z 169.477,A -85,B 0,C 180,E1 34235.937,E2 34235.937} C_VEL
LIN {X 0,Y 735.992,Z 169.48,A -85,B 0,C 180,E1 34233.569,E2 34233.569} C_VEL
LIN {X 0,Y 736.042,Z 169.482,A -85,B 0,C 180,E1 34230.988,E2 34230.988} C_VEL
LIN {X 0,Y 736.012,Z 169.474,A -85,B 0,C 180,E1 34228.126,E2 34228.126} C_VEL
LIN {X 0,Y 735.993,Z 169.48,A -85,B 0,C 180,E1 34225.763,E2 34225.763} C_VEL
LIN {X 0,Y 736.012,Z 169.482,A -85,B 0,C 180,E1 34223.33,E2 34223.33} C_VEL
LIN {X 0,Y 736.018,Z 169.482,A -85,B 0,C 180,E1 34220.269,E2 34220.269} C_VEL
LIN {X 0,Y 735.992,Z 169.481,A -85,B 0,C 180,E1 34217.881,E2 34217.881} C_VEL
LIN {X 0,Y 736.001,Z 169.481,A -85,B 0,C 180,E1 34215.524,E2 34215.524} C_VEL
LIN {X 0,Y 736.072,Z 169.48,A -85,B 0,C 180,E1 34212.713,E2 34212.713} C_VEL
LIN {X 0,Y 735.994,Z 169.482,A -85,B 0,C 180,E1 34209.997,E2 34209.997} C_VEL
LIN {X 0,Y 736,Z 169.48,A -85,B 0,C 180,E1 34207.651,E2 34207.651} C_VEL
LIN {X 0,Y 736.075,Z 169.482,A -85,B 0,C 180,E1 34204.831,E2 34204.831} C_VEL
LIN {X 0,Y 735.996,Z 169.48,A -85,B 0,C 180,E1 34202.18,E2 34202.18} C_VEL
LIN {X 0,Y 735.993,Z 169.482,A -85,B 0,C 180,E1 34199.922,E2 34199.922} C_VEL
LIN {X 0,Y 736.032,Z 169.481,A -85,B 0,C 180,E1 34197.431,E2 34197.431} C_VEL
LIN {X 0,Y 736.01,Z 169.481,A -85,B 0,C 180,E1 34194.465,E2 34194.465} C_VEL
LIN {X 0,Y 735.993,Z 169.479,A -85,B 0,C 180,E1 34192.113,E2 34192.113} C_VEL
LIN {X 0,Y 736.016,Z 169.482,A -85,B 0,C 180,E1 34189.67,E2 34189.67} C_VEL
LIN {X 0,Y 736.02,Z 169.481,A -85,B 0,C 180,E1 34186.647,E2 34186.647} C_VEL
LIN {X 0,Y 735.993,Z 169.482,A -85,B 0,C 180,E1 34184.234,E2 34184.234} C_VEL
LIN {X 0,Y 736.012,Z 169.48,A -85,B 0,C 180,E1 34181.792,E2 34181.792} C_VEL
LIN {X 0,Y 736.018,Z 169.48,A -85,B 0,C 180,E1 34178.719,E2 34178.719} C_VEL
LIN {X 0,Y 735.994,Z 169.482,A -85,B 0,C 180,E1 34176.283,E2 34176.283} C_VEL
LIN {X 0,Y 736.02,Z 169.481,A -85,B 0,C 180,E1 34173.799,E2 34173.799} C_VEL
LIN {X 0,Y 736.018,Z 169.479,A -85,B 0,C 180,E1 34170.81,E2 34170.81} C_VEL
LIN {X 0,Y 735.995,Z 169.482,A -85,B 0,C 180,E1 34168.463,E2 34168.463} C_VEL
LIN {X 0,Y 736.005,Z 169.481,A -85,B 0,C 180,E1 34166.057,E2 34166.057} C_VEL
LIN {X 0,Y 736.059,Z 169.482,A -85,B 0,C 180,E1 34163.196,E2 34163.196} C_VEL
LIN {X 0,Y 735.997,Z 169.479,A -85,B 0,C 180,E1 34160.616,E2 34160.616} C_VEL
LIN {X 0,Y 735.998,Z 169.482,A -85,B 0,C 180,E1 34158.264,E2 34158.264} C_VEL
LIN {X 0,Y 736.09,Z 169.48,A -85,B 0,C 180,E1 34155.484,E2 34155.484} C_VEL
LIN {X 0,Y 735.997,Z 169.48,A -85,B 0,C 180,E1 34152.694,E2 34152.694} C_VEL
LIN {X 0,Y 735.997,Z 169.483,A -85,B 0,C 180,E1 34150.386,E2 34150.386} C_VEL
LIN {X 0,Y 736.092,Z 169.471,A -85,B 0,C 180,E1 34147.577,E2 34147.577} C_VEL
LIN {X 0,Y 735.996,Z 169.483,A -85,B 0,C 180,E1 34144.786,E2 34144.786} C_VEL
LIN {X 0,Y 735.997,Z 169.476,A -85,B 0,C 180,E1 34142.449,E2 34142.449} C_VEL
LIN {X 0,Y 736.032,Z 169.753,A -85,B 0,C 180,E1 34140.621,E2 34140.621} C_VEL
LIN {X 0,Y 737.653,Z 175.855,A -85,B 0,C 180,E1 34140.052,E2 34140.052} C_VEL
LIN {X 0,Y 737.332,Z 212.213,A -85,B 0,C 180,E1 34137.233,E2 34137.233} C_VEL
LIN {X 0,Y 737.331,Z 226.556,A -85,B 0,C 180,E1 34136.164,E2 34136.164} C_VEL
LIN {X 0,Y 738.229,Z 231.976,A -85,B 0,C 180,E1 34136.067,E2 34136.067} C_VEL
LIN {X 0,Y 737.774,Z 504.998,A -85,B 0,C 180,E1 34133.219,E2 34133.219} C_VEL
LIN {X 0,Y 737.675,Z 534.583,A -85,B 0,C 180,E1 34132.869,E2 34132.869} C_VEL
LIN {X 0,Y 737.569,Z 556.452,A -85,B 0,C 180,E1 34132.462,E2 34132.462} C_VEL
LIN {X 0,Y 737.416,Z 576.362,A -85,B 0,C 180,E1 34131.957,E2 34131.957} C_VEL
LIN {X 0,Y 737.248,Z 597.295,A -85,B 0,C 180,E1 34131.291,E2 34131.291} C_VEL
LIN {X 0,Y 737.083,Z 618.332,A -85,B 0,C 180,E1 34130.458,E2 34130.458} C_VEL
LIN {X 0,Y 736.887,Z 636.749,A -85,B 0,C 180,E1 34129.579,E2 34129.579} C_VEL
LIN {X 0,Y 736.701,Z 655.336,A -85,B 0,C 180,E1 34128.546,E2 34128.546} C_VEL
LIN {X 0,Y 736.528,Z 673.824,A -85,B 0,C 180,E1 34127.334,E2 34127.334} C_VEL
LIN {X 0,Y 736.382,Z 689.723,A -85,B 0,C 180,E1 34126.119,E2 34126.119} C_VEL
LIN {X 0,Y 736.238,Z 705.013,A -85,B 0,C 180,E1 34124.765,E2 34124.765} C_VEL
LIN {X 0,Y 736.116,Z 719.459,A -85,B 0,C 180,E1 34123.269,E2 34123.269} C_VEL
LIN {X 0,Y 736.052,Z 731.341,A -85,B 0,C 180,E1 34121.835,E2 34121.835} C_VEL
LIN {X 0,Y 735.991,Z 742.376,A -85,B 0,C 180,E1 34120.25,E2 34120.25} C_VEL
LIN {X 0,Y 735.939,Z 751.887,A -85,B 0,C 180,E1 34118.594,E2 34118.594} C_VEL
LIN {X 0,Y 735.92,Z 759.569,A -85,B 0,C 180,E1 34116.944,E2 34116.944} C_VEL
LIN {X 0,Y 735.917,Z 765.419,A -85,B 0,C 180,E1 34115.3,E2 34115.3} C_VEL
LIN {X 0,Y 735.916,Z 769.785,A -85,B 0,C 180,E1 34113.583,E2 34113.583} C_VEL
LIN {X 0,Y 735.919,Z 772.491,A -85,B 0,C 180,E1 34111.868,E2 34111.868} C_VEL
LIN {X 0,Y 735.913,Z 773.484,A -85,B 0,C 180,E1 34110.078,E2 34110.078} C_VEL
LIN {X 0,Y 735.907,Z 772.691,A -85,B 0,C 180,E1 34108.365,E2 34108.365} C_VEL
LIN {X 0,Y 735.908,Z 770.101,A -85,B 0,C 180,E1 34106.573,E2 34106.573} C_VEL
LIN {X 0,Y 735.905,Z 766.161,A -85,B 0,C 180,E1 34104.934,E2 34104.934} C_VEL
LIN {X 0,Y 735.913,Z 760.174,A -85,B 0,C 180,E1 34103.212,E2 34103.212} C_VEL
LIN {X 0,Y 735.936,Z 752.567,A -85,B 0,C 180,E1 34101.538,E2 34101.538} C_VEL
LIN {X 0,Y 735.991,Z 743.899,A -85,B 0,C 180,E1 34099.987,E2 34099.987} C_VEL
LIN {X 0,Y 736.039,Z 732.527,A -85,B 0,C 180,E1 34098.324,E2 34098.324} C_VEL
LIN {X 0,Y 736.113,Z 720.164,A -85,B 0,C 180,E1 34096.811,E2 34096.811} C_VEL
LIN {X 0,Y 736.23,Z 706.444,A -85,B 0,C 180,E1 34095.37,E2 34095.37} C_VEL
LIN {X 0,Y 736.373,Z 690.717,A -85,B 0,C 180,E1 34093.961,E2 34093.961} C_VEL
LIN {X 0,Y 736.509,Z 674.948,A -85,B 0,C 180,E1 34092.747,E2 34092.747} C_VEL
LIN {X 0,Y 736.68,Z 657.163,A -85,B 0,C 180,E1 34091.566,E2 34091.566} C_VEL
LIN {X 0,Y 736.879,Z 637.904,A -85,B 0,C 180,E1 34090.48,E2 34090.48} C_VEL
LIN {X 0,Y 737.062,Z 619.605,A -85,B 0,C 180,E1 34089.599,E2 34089.599} C_VEL
LIN {X 0,Y 737.226,Z 599.016,A -85,B 0,C 180,E1 34088.772,E2 34088.772} C_VEL
LIN {X 0,Y 737.41,Z 577.88,A -85,B 0,C 180,E1 34088.086,E2 34088.086} C_VEL
LIN {X 0,Y 737.552,Z 557.778,A -85,B 0,C 180,E1 34087.568,E2 34087.568} C_VEL
LIN {X 0,Y 737.669,Z 536.323,A -85,B 0,C 180,E1 34087.159,E2 34087.159} C_VEL
LIN {X 0,Y 737.769,Z 508.304,A -85,B 0,C 180,E1 34086.815,E2 34086.815} C_VEL
LIN {X 0,Y 738.221,Z 236.299,A -85,B 0,C 180,E1 34083.979,E2 34083.979} C_VEL
LIN {X 0,Y 737.976,Z 229.538,A -85,B 0,C 180,E1 34083.898,E2 34083.898} C_VEL
LIN {X 0,Y 737.277,Z 225.847,A -85,B 0,C 180,E1 34083.8,E2 34083.8} C_VEL
LIN {X 0,Y 737.552,Z 187.785,A -85,B 0,C 180,E1 34080.881,E2 34080.881} C_VEL
LIN {X 0,Y 737.582,Z 174.925,A -85,B 0,C 180,E1 34079.871,E2 34079.871} C_VEL
LIN {X 0,Y 736.008,Z 169.595,A -85,B 0,C 180,E1 34079.347,E2 34079.347} C_VEL
LIN {X 0,Y 736.015,Z 169.472,A -85,B 0,C 180,E1 34076.904,E2 34076.904} C_VEL
LIN {X 0,Y 736.02,Z 169.48,A -85,B 0,C 180,E1 34073.878,E2 34073.878} C_VEL
LIN {X 0,Y 735.994,Z 169.478,A -85,B 0,C 180,E1 34071.493,E2 34071.493} C_VEL
LIN {X 0,Y 736.001,Z 169.483,A -85,B 0,C 180,E1 34069.175,E2 34069.175} C_VEL
LIN {X 0,Y 736.081,Z 169.482,A -85,B 0,C 180,E1 34066.372,E2 34066.372} C_VEL
LIN {X 0,Y 735.995,Z 169.481,A -85,B 0,C 180,E1 34063.642,E2 34063.642} C_VEL
LIN {X 0,Y 735.998,Z 169.482,A -85,B 0,C 180,E1 34061.308,E2 34061.308} C_VEL
LIN {X 0,Y 736.084,Z 169.482,A -85,B 0,C 180,E1 34058.473,E2 34058.473} C_VEL
LIN {X 0,Y 735.995,Z 169.48,A -85,B 0,C 180,E1 34055.745,E2 34055.745} C_VEL
LIN {X 0,Y 735.999,Z 169.481,A -85,B 0,C 180,E1 34053.382,E2 34053.382} C_VEL
LIN {X 0,Y 736.078,Z 169.479,A -85,B 0,C 180,E1 34050.534,E2 34050.534} C_VEL
LIN {X 0,Y 735.996,Z 169.476,A -85,B 0,C 180,E1 34047.862,E2 34047.862} C_VEL
LIN {X 0,Y 735.998,Z 169.481,A -85,B 0,C 180,E1 34045.51,E2 34045.51} C_VEL
LIN {X 0,Y 736.092,Z 169.48,A -85,B 0,C 180,E1 34042.692,E2 34042.692} C_VEL
LIN {X 0,Y 735.995,Z 169.482,A -85,B 0,C 180,E1 34039.938,E2 34039.938} C_VEL
LIN {X 0,Y 735.996,Z 169.48,A -85,B 0,C 180,E1 34037.635,E2 34037.635} C_VEL
LIN {X 0,Y 736.091,Z 169.481,A -85,B 0,C 180,E1 34034.876,E2 34034.876} C_VEL
LIN {X 0,Y 735.997,Z 169.481,A -85,B 0,C 180,E1 34032.034,E2 34032.034} C_VEL
LIN {X 0,Y 736,Z 169.481,A -85,B 0,C 180,E1 34029.619,E2 34029.619} C_VEL
LIN {X 0,Y 736.076,Z 169.482,A -85,B 0,C 180,E1 34026.787,E2 34026.787} C_VEL
LIN {X 0,Y 735.996,Z 169.481,A -85,B 0,C 180,E1 34024.129,E2 34024.129} C_VEL
LIN {X 0,Y 735.996,Z 169.481,A -85,B 0,C 180,E1 34021.791,E2 34021.791} C_VEL
LIN {X 0,Y 736.088,Z 169.482,A -85,B 0,C 180,E1 34019.066,E2 34019.066} C_VEL
LIN {X 0,Y 735.997,Z 169.482,A -85,B 0,C 180,E1 34016.261,E2 34016.261} C_VEL
LIN {X 0,Y 735.995,Z 169.481,A -85,B 0,C 180,E1 34013.894,E2 34013.894} C_VEL
LIN {X 0,Y 736.07,Z 169.48,A -85,B 0,C 180,E1 34011.249,E2 34011.249} C_VEL
LIN {X 0,Y 736.07,Z 169.48,A -85,B 0,C 180,E1 34008.96,E2 34008.96} C_VEL
LIN {X 0,Y 735.025,Z 169.603,A -85,B 0,C 180,E1 34008.361,E2 34008.361} C_VEL
LIN {X 0,Y 728.587,Z 170.41,A -85,B 0,C 180,E1 34006.681,E2 34006.681} C_VEL
LIN {X 0,Y 728.054,Z 170.471,A -85,B 0,C 180,E1 34006.245,E2 34006.245} C_VEL
LIN {X 0,Y 728.061,Z 170.47,A -85,B 0,C 180,E1 34003.894,E2 34003.894} C_VEL
LIN {X 0,Y 728.123,Z 170.471,A -85,B 0,C 180,E1 34001.007,E2 34001.007} C_VEL
LIN {X 0,Y 728.056,Z 170.469,A -85,B 0,C 180,E1 33998.379,E2 33998.379} C_VEL
LIN {X 0,Y 728.061,Z 170.471,A -85,B 0,C 180,E1 33996.014,E2 33996.014} C_VEL
LIN {X 0,Y 728.13,Z 170.462,A -85,B 0,C 180,E1 33993.141,E2 33993.141} C_VEL
LIN {X 0,Y 728.056,Z 170.469,A -85,B 0,C 180,E1 33990.459,E2 33990.459} C_VEL
LIN {X 0,Y 728.057,Z 170.471,A -85,B 0,C 180,E1 33988.172,E2 33988.172} C_VEL
LIN {X 0,Y 728.146,Z 170.463,A -85,B 0,C 180,E1 33985.329,E2 33985.329} C_VEL
LIN {X 0,Y 728.057,Z 170.471,A -85,B 0,C 180,E1 33982.625,E2 33982.625} C_VEL
LIN {X 0,Y 728.057,Z 170.471,A -85,B 0,C 180,E1 33980.262,E2 33980.262} C_VEL
LIN {X 0,Y 728.148,Z 170.472,A -85,B 0,C 180,E1 33977.498,E2 33977.498} C_VEL
LIN {X 0,Y 728.061,Z 170.472,A -85,B 0,C 180,E1 33974.763,E2 33974.763} C_VEL
LIN {X 0,Y 728.055,Z 170.471,A -85,B 0,C 180,E1 33972.395,E2 33972.395} C_VEL
LIN {X 0,Y 728.126,Z 170.471,A -85,B 0,C 180,E1 33969.734,E2 33969.734} C_VEL
LIN {X 0,Y 728.062,Z 170.471,A -85,B 0,C 180,E1 33966.875,E2 33966.875} C_VEL
LIN {X 0,Y 728.057,Z 170.471,A -85,B 0,C 180,E1 33964.454,E2 33964.454} C_VEL
LIN {X 0,Y 728.146,Z 170.472,A -85,B 0,C 180,E1 33961.634,E2 33961.634} C_VEL
LIN {X 0,Y 728.058,Z 170.472,A -85,B 0,C 180,E1 33958.905,E2 33958.905} C_VEL
LIN {X 0,Y 728.058,Z 170.471,A -85,B 0,C 180,E1 33956.505,E2 33956.505} C_VEL
LIN {X 0,Y 728.143,Z 170.472,A -85,B 0,C 180,E1 33953.661,E2 33953.661} C_VEL
LIN {X 0,Y 728.056,Z 170.472,A -85,B 0,C 180,E1 33950.918,E2 33950.918} C_VEL
LIN {X 0,Y 728.058,Z 170.472,A -85,B 0,C 180,E1 33948.577,E2 33948.577} C_VEL
LIN {X 0,Y 728.145,Z 170.472,A -85,B 0,C 180,E1 33945.775,E2 33945.775} C_VEL
LIN {X 0,Y 728.056,Z 170.471,A -85,B 0,C 180,E1 33943.015,E2 33943.015} C_VEL
LIN {X 0,Y 728.057,Z 170.472,A -85,B 0,C 180,E1 33940.683,E2 33940.683} C_VEL
LIN {X 0,Y 728.151,Z 170.471,A -85,B 0,C 180,E1 33937.892,E2 33937.892} C_VEL
LIN {X 0,Y 728.056,Z 170.472,A -85,B 0,C 180,E1 33935.121,E2 33935.121} C_VEL
LIN {X 0,Y 728.057,Z 170.472,A -85,B 0,C 180,E1 33932.755,E2 33932.755} C_VEL
LIN {X 0,Y 728.144,Z 170.471,A -85,B 0,C 180,E1 33929.921,E2 33929.921} C_VEL
LIN {X 0,Y 728.054,Z 170.472,A -85,B 0,C 180,E1 33927.166,E2 33927.166} C_VEL
LIN {X 0,Y 728.06,Z 170.472,A -85,B 0,C 180,E1 33924.8,E2 33924.8} C_VEL
LIN {X 0,Y 728.132,Z 170.472,A -85,B 0,C 180,E1 33921.949,E2 33921.949} C_VEL
LIN {X 0,Y 728.054,Z 170.472,A -85,B 0,C 180,E1 33919.237,E2 33919.237} C_VEL
LIN {X 0,Y 728.063,Z 170.471,A -85,B 0,C 180,E1 33916.834,E2 33916.834} C_VEL
LIN {X 0,Y 728.122,Z 170.472,A -85,B 0,C 180,E1 33913.979,E2 33913.979} C_VEL
LIN {X 0,Y 728.055,Z 170.472,A -85,B 0,C 180,E1 33911.34,E2 33911.34} C_VEL
LIN {X 0,Y 728.06,Z 170.472,A -85,B 0,C 180,E1 33908.998,E2 33908.998} C_VEL
LIN {X 0,Y 728.136,Z 170.472,A -85,B 0,C 180,E1 33906.144,E2 33906.144} C_VEL
LIN {X 0,Y 728.055,Z 170.471,A -85,B 0,C 180,E1 33903.407,E2 33903.407} C_VEL
LIN {X 0,Y 728.064,Z 170.472,A -85,B 0,C 180,E1 33901.005,E2 33901.005} C_VEL
LIN {X 0,Y 728.127,Z 170.472,A -85,B 0,C 180,E1 33898.18,E2 33898.18} C_VEL
LIN {X 0,Y 728.055,Z 170.472,A -85,B 0,C 180,E1 33895.49,E2 33895.49} C_VEL
LIN {X 0,Y 728.07,Z 170.471,A -85,B 0,C 180,E1 33893.027,E2 33893.027} C_VEL
LIN {X 0,Y 728.089,Z 170.471,A -85,B 0,C 180,E1 33890.013,E2 33890.013} C_VEL
LIN {X 0,Y 728.053,Z 170.471,A -85,B 0,C 180,E1 33887.519,E2 33887.519} C_VEL
LIN {X 0,Y 728.07,Z 170.472,A -85,B 0,C 180,E1 33885.106,E2 33885.106} C_VEL
LIN {X 0,Y 728.086,Z 170.471,A -85,B 0,C 180,E1 33882.081,E2 33882.081} C_VEL
LIN {X 0,Y 728.054,Z 170.471,A -85,B 0,C 180,E1 33879.614,E2 33879.614} C_VEL
LIN {X 0,Y 728.071,Z 170.471,A -85,B 0,C 180,E1 33877.177,E2 33877.177} C_VEL
LIN {X 0,Y 728.075,Z 170.468,A -85,B 0,C 180,E1 33874.078,E2 33874.078} C_VEL
LIN {X 0,Y 728.053,Z 170.471,A -85,B 0,C 180,E1 33871.638,E2 33871.638} C_VEL
LIN {X 0,Y 728.071,Z 170.469,A -85,B 0,C 180,E1 33869.269,E2 33869.269} C_VEL
LIN {X 0,Y 728.085,Z 170.468,A -85,B 0,C 180,E1 33866.245,E2 33866.245} C_VEL
LIN {X 0,Y 728.055,Z 170.471,A -85,B 0,C 180,E1 33863.728,E2 33863.728} C_VEL
LIN {X 0,Y 728.082,Z 170.469,A -85,B 0,C 180,E1 33861.257,E2 33861.257} C_VEL
LIN {X 0,Y 728.075,Z 170.47,A -85,B 0,C 180,E1 33858.247,E2 33858.247} C_VEL
LIN {X 0,Y 728.053,Z 170.47,A -85,B 0,C 180,E1 33855.779,E2 33855.779} C_VEL
LIN {X 0,Y 728.093,Z 170.47,A -85,B 0,C 180,E1 33853.258,E2 33853.258} C_VEL
LIN {X 0,Y 728.071,Z 170.471,A -85,B 0,C 180,E1 33850.284,E2 33850.284} C_VEL
LIN {X 0,Y 728.054,Z 170.469,A -85,B 0,C 180,E1 33847.894,E2 33847.894} C_VEL
LIN {X 0,Y 728.073,Z 170.47,A -85,B 0,C 180,E1 33845.517,E2 33845.517} C_VEL
LIN {X 0,Y 728.076,Z 170.468,A -85,B 0,C 180,E1 33842.44,E2 33842.44} C_VEL
LIN {X 0,Y 728.054,Z 170.471,A -85,B 0,C 180,E1 33840.079,E2 33840.079} C_VEL
LIN {X 0,Y 728.064,Z 170.47,A -85,B 0,C 180,E1 33837.717,E2 33837.717} C_VEL
LIN {X 0,Y 728.112,Z 170.47,A -85,B 0,C 180,E1 33834.8,E2 33834.8} C_VEL
LIN {X 0,Y 728.057,Z 170.467,A -85,B 0,C 180,E1 33832.265,E2 33832.265} C_VEL
LIN {X 0,Y 728.061,Z 170.47,A -85,B 0,C 180,E1 33829.875,E2 33829.875} C_VEL
LIN {X 0,Y 728.141,Z 170.47,A -85,B 0,C 180,E1 33827.066,E2 33827.066} C_VEL
LIN {X 0,Y 728.059,Z 170.471,A -85,B 0,C 180,E1 33824.384,E2 33824.384} C_VEL
LIN {X 0,Y 728.059,Z 170.468,A -85,B 0,C 180,E1 33822,E2 33822} C_VEL
LIN {X 0,Y 728.152,Z 170.47,A -85,B 0,C 180,E1 33819.23,E2 33819.23} C_VEL
LIN {X 0,Y 728.058,Z 170.471,A -85,B 0,C 180,E1 33816.444,E2 33816.444} C_VEL
LIN {X 0,Y 728.064,Z 170.47,A -85,B 0,C 180,E1 33814.017,E2 33814.017} C_VEL
LIN {X 0,Y 728.13,Z 170.467,A -85,B 0,C 180,E1 33811.164,E2 33811.164} C_VEL
LIN {X 0,Y 728.058,Z 170.471,A -85,B 0,C 180,E1 33808.511,E2 33808.511} C_VEL
LIN {X 0,Y 728.063,Z 170.469,A -85,B 0,C 180,E1 33806.111,E2 33806.111} C_VEL
LIN {X 0,Y 728.14,Z 170.471,A -85,B 0,C 180,E1 33803.307,E2 33803.307} C_VEL
LIN {X 0,Y 728.058,Z 170.468,A -85,B 0,C 180,E1 33800.617,E2 33800.617} C_VEL
LIN {X 0,Y 728.063,Z 170.471,A -85,B 0,C 180,E1 33798.213,E2 33798.213} C_VEL
LIN {X 0,Y 728.145,Z 170.469,A -85,B 0,C 180,E1 33795.436,E2 33795.436} C_VEL
LIN {X 0,Y 728.059,Z 170.469,A -85,B 0,C 180,E1 33792.714,E2 33792.714} C_VEL
LIN {X 0,Y 728.058,Z 170.472,A -85,B 0,C 180,E1 33790.401,E2 33790.401} C_VEL
LIN {X 0,Y 728.152,Z 170.457,A -85,B 0,C 180,E1 33787.596,E2 33787.596} C_VEL
LIN {X 0,Y 728.058,Z 170.472,A -85,B 0,C 180,E1 33784.787,E2 33784.787} C_VEL
LIN {X 0,Y 728.063,Z 170.462,A -85,B 0,C 180,E1 33782.369,E2 33782.369} C_VEL
LIN {X 0,Y 728.101,Z 170.751,A -85,B 0,C 180,E1 33780.911,E2 33780.911} C_VEL
LIN {X 0,Y 730.235,Z 178.696,A -85,B 0,C 180,E1 33780.162,E2 33780.162} C_VEL
LIN {X 0,Y 729.817,Z 214.429,A -85,B 0,C 180,E1 33777.365,E2 33777.365} C_VEL
LIN {X 0,Y 729.795,Z 226.493,A -85,B 0,C 180,E1 33776.456,E2 33776.456} C_VEL
LIN {X 0,Y 731.036,Z 233.293,A -85,B 0,C 180,E1 33776.328,E2 33776.328} C_VEL
LIN {X 0,Y 730.417,Z 506.271,A -85,B 0,C 180,E1 33773.453,E2 33773.453} C_VEL
LIN {X 0,Y 730.287,Z 535.419,A -85,B 0,C 180,E1 33773.1,E2 33773.1} C_VEL
LIN {X 0,Y 730.139,Z 556.911,A -85,B 0,C 180,E1 33772.691,E2 33772.691} C_VEL
LIN {X 0,Y 729.942,Z 576.835,A -85,B 0,C 180,E1 33772.18,E2 33772.18} C_VEL
LIN {X 0,Y 729.717,Z 597.82,A -85,B 0,C 180,E1 33771.503,E2 33771.503} C_VEL
LIN {X 0,Y 729.483,Z 618.85,A -85,B 0,C 180,E1 33770.657,E2 33770.657} C_VEL
LIN {X 0,Y 729.226,Z 636.744,A -85,B 0,C 180,E1 33769.793,E2 33769.793} C_VEL
LIN {X 0,Y 728.995,Z 655.188,A -85,B 0,C 180,E1 33768.759,E2 33768.759} C_VEL
LIN {X 0,Y 728.75,Z 673.827,A -85,B 0,C 180,E1 33767.524,E2 33767.524} C_VEL
LIN {X 0,Y 728.543,Z 689.715,A -85,B 0,C 180,E1 33766.298,E2 33766.298} C_VEL
LIN {X 0,Y 728.361,Z 704.751,A -85,B 0,C 180,E1 33764.954,E2 33764.954} C_VEL
LIN {X 0,Y 728.197,Z 719.459,A -85,B 0,C 180,E1 33763.416,E2 33763.416} C_VEL
LIN {X 0,Y 728.107,Z 731.333,A -85,B 0,C 180,E1 33761.966,E2 33761.966} C_VEL
LIN {X 0,Y 728.022,Z 742.379,A -85,B 0,C 180,E1 33760.364,E2 33760.364} C_VEL
LIN {X 0,Y 727.956,Z 751.889,A -85,B 0,C 180,E1 33758.689,E2 33758.689} C_VEL
LIN {X 0,Y 727.94,Z 759.24,A -85,B 0,C 180,E1 33757.1,E2 33757.1} C_VEL
LIN {X 0,Y 727.922,Z 765.168,A -85,B 0,C 180,E1 33755.438,E2 33755.438} C_VEL
LIN {X 0,Y 727.917,Z 769.787,A -85,B 0,C 180,E1 33753.622,E2 33753.622} C_VEL
LIN {X 0,Y 727.919,Z 772.488,A -85,B 0,C 180,E1 33751.889,E2 33751.889} C_VEL
LIN {X 0,Y 727.913,Z 773.484,A -85,B 0,C 180,E1 33750.079,E2 33750.079} C_VEL
LIN {X 0,Y 727.913,Z 772.628,A -85,B 0,C 180,E1 33748.268,E2 33748.268} C_VEL
LIN {X 0,Y 727.911,Z 770.102,A -85,B 0,C 180,E1 33746.535,E2 33746.535} C_VEL
LIN {X 0,Y 727.913,Z 765.927,A -85,B 0,C 180,E1 33744.799,E2 33744.799} C_VEL
LIN {X 0,Y 727.925,Z 759.875,A -85,B 0,C 180,E1 33743.058,E2 33743.058} C_VEL
LIN {X 0,Y 727.952,Z 752.295,A -85,B 0,C 180,E1 33741.391,E2 33741.391} C_VEL
LIN {X 0,Y 728.017,Z 743.413,A -85,B 0,C 180,E1 33739.796,E2 33739.796} C_VEL
LIN {X 0,Y 728.101,Z 731.947,A -85,B 0,C 180,E1 33738.114,E2 33738.114} C_VEL
LIN {X 0,Y 728.188,Z 720.164,A -85,B 0,C 180,E1 33736.665,E2 33736.665} C_VEL
LIN {X 0,Y 728.346,Z 706.448,A -85,B 0,C 180,E1 33735.208,E2 33735.208} C_VEL
LIN {X 0,Y 728.538,Z 690.709,A -85,B 0,C 180,E1 33733.784,E2 33733.784} C_VEL
LIN {X 0,Y 728.73,Z 674.932,A -85,B 0,C 180,E1 33732.557,E2 33732.557} C_VEL
LIN {X 0,Y 728.957,Z 657.17,A -85,B 0,C 180,E1 33731.364,E2 33731.364} C_VEL
LIN {X 0,Y 729.215,Z 638.348,A -85,B 0,C 180,E1 33730.29,E2 33730.29} C_VEL
LIN {X 0,Y 729.449,Z 620.709,A -85,B 0,C 180,E1 33729.427,E2 33729.427} C_VEL
LIN {X 0,Y 729.674,Z 601.266,A -85,B 0,C 180,E1 33728.626,E2 33728.626} C_VEL
LIN {X 0,Y 729.928,Z 579.419,A -85,B 0,C 180,E1 33727.894,E2 33727.894} C_VEL
LIN {X 0,Y 730.108,Z 559.236,A -85,B 0,C 180,E1 33727.362,E2 33727.362} C_VEL
LIN {X 0,Y 730.278,Z 537.645,A -85,B 0,C 180,E1 33726.936,E2 33726.936} C_VEL
LIN {X 0,Y 730.405,Z 510.848,A -85,B 0,C 180,E1 33726.594,E2 33726.594} C_VEL
LIN {X 0,Y 731.021,Z 239.734,A -85,B 0,C 180,E1 33723.74,E2 33723.74} C_VEL
LIN {X 0,Y 730.805,Z 231.021,A -85,B 0,C 180,E1 33723.638,E2 33723.638} C_VEL
LIN {X 0,Y 729.755,Z 225.975,A -85,B 0,C 180,E1 33723.517,E2 33723.517} C_VEL
LIN {X 0,Y 730.127,Z 188.012,A -85,B 0,C 180,E1 33720.574,E2 33720.574} C_VEL
LIN {X 0,Y 730.159,Z 177.559,A -85,B 0,C 180,E1 33719.743,E2 33719.743} C_VEL
LIN {X 0,Y 728.078,Z 170.579,A -85,B 0,C 180,E1 33719.053,E2 33719.053} C_VEL
LIN {X 0,Y 728.126,Z 170.462,A -85,B 0,C 180,E1 33716.182,E2 33716.182} C_VEL
LIN {X 0,Y 728.056,Z 170.468,A -85,B 0,C 180,E1 33713.517,E2 33713.517} C_VEL
LIN {X 0,Y 728.063,Z 170.466,A -85,B 0,C 180,E1 33711.131,E2 33711.131} C_VEL
LIN {X 0,Y 728.122,Z 170.47,A -85,B 0,C 180,E1 33708.246,E2 33708.246} C_VEL
LIN {X 0,Y 728.058,Z 170.471,A -85,B 0,C 180,E1 33705.657,E2 33705.657} C_VEL
LIN {X 0,Y 728.061,Z 170.47,A -85,B 0,C 180,E1 33703.26,E2 33703.26} C_VEL
LIN {X 0,Y 728.134,Z 170.468,A -85,B 0,C 180,E1 33700.403,E2 33700.403} C_VEL
LIN {X 0,Y 728.058,Z 170.471,A -85,B 0,C 180,E1 33697.726,E2 33697.726} C_VEL
LIN {X 0,Y 728.062,Z 170.468,A -85,B 0,C 180,E1 33695.347,E2 33695.347} C_VEL
LIN {X 0,Y 728.132,Z 170.471,A -85,B 0,C 180,E1 33692.475,E2 33692.475} C_VEL
LIN {X 0,Y 728.056,Z 170.467,A -85,B 0,C 180,E1 33689.79,E2 33689.79} C_VEL
LIN {X 0,Y 728.058,Z 170.464,A -85,B 0,C 180,E1 33687.481,E2 33687.481} C_VEL
LIN {X 0,Y 728.147,Z 170.472,A -85,B 0,C 180,E1 33684.674,E2 33684.674} C_VEL
LIN {X 0,Y 728.058,Z 170.469,A -85,B 0,C 180,E1 33681.935,E2 33681.935} C_VEL
LIN {X 0,Y 728.058,Z 170.471,A -85,B 0,C 180,E1 33679.579,E2 33679.579} C_VEL
LIN {X 0,Y 728.147,Z 170.47,A -85,B 0,C 180,E1 33676.761,E2 33676.761} C_VEL
LIN {X 0,Y 728.06,Z 170.469,A -85,B 0,C 180,E1 33674.069,E2 33674.069} C_VEL
LIN {X 0,Y 728.056,Z 170.47,A -85,B 0,C 180,E1 33671.728,E2 33671.728} C_VEL
LIN {X 0,Y 728.148,Z 170.47,A -85,B 0,C 180,E1 33668.927,E2 33668.927} C_VEL
LIN {X 0,Y 728.059,Z 170.471,A -85,B 0,C 180,E1 33666.15,E2 33666.15} C_VEL
LIN {X 0,Y 728.057,Z 170.47,A -85,B 0,C 180,E1 33663.78,E2 33663.78} C_VEL
LIN {X 0,Y 728.152,Z 170.47,A -85,B 0,C 180,E1 33661.023,E2 33661.023} C_VEL
LIN {X 0,Y 728.06,Z 170.468,A -85,B 0,C 180,E1 33658.269,E2 33658.269} C_VEL
LIN {X 0,Y 728.054,Z 170.471,A -85,B 0,C 180,E1 33655.905,E2 33655.905} C_VEL
LIN {X 0,Y 728.148,Z 170.47,A -85,B 0,C 180,E1 33653.139,E2 33653.139} C_VEL
LIN {X 0,Y 728.061,Z 170.471,A -85,B 0,C 180,E1 33650.355,E2 33650.355} C_VEL
LIN {X 0,Y 728.058,Z 170.468,A -85,B 0,C 180,E1 33647.951,E2 33647.951} C_VEL
LIN {X 0,Y 728.054,Z 170.471,A -85,B 0,C 180,E1 33646.245,E2 33646.245} C_VEL
LIN {X 0,Y 727.051,Z 170.6,A -85,B 0,C 180,E1 33645.639,E2 33645.639} C_VEL
LIN {X 0,Y 720.744,Z 171.383,A -85,B 0,C 180,E1 33643.984,E2 33643.984} C_VEL
LIN {X 0,Y 720.164,Z 171.459,A -85,B 0,C 180,E1 33643.499,E2 33643.499} C_VEL
LIN {X 0,Y 720.133,Z 171.46,A -85,B 0,C 180,E1 33640.619,E2 33640.619} C_VEL
LIN {X 0,Y 720.115,Z 171.458,A -85,B 0,C 180,E1 33638.239,E2 33638.239} C_VEL
LIN {X 0,Y 720.146,Z 171.46,A -85,B 0,C 180,E1 33635.733,E2 33635.733} C_VEL
LIN {X 0,Y 720.13,Z 171.448,A -85,B 0,C 180,E1 33632.686,E2 33632.686} C_VEL
LIN {X 0,Y 720.116,Z 171.457,A -85,B 0,C 180,E1 33630.284,E2 33630.284} C_VEL
LIN {X 0,Y 720.159,Z 171.46,A -85,B 0,C 180,E1 33627.719,E2 33627.719} C_VEL
LIN {X 0,Y 720.131,Z 171.453,A -85,B 0,C 180,E1 33624.815,E2 33624.815} C_VEL
LIN {X 0,Y 720.115,Z 171.46,A -85,B 0,C 180,E1 33622.442,E2 33622.442} C_VEL
LIN {X 0,Y 720.137,Z 171.46,A -85,B 0,C 180,E1 33619.994,E2 33619.994} C_VEL
LIN {X 0,Y 720.136,Z 171.46,A -85,B 0,C 180,E1 33616.906,E2 33616.906} C_VEL
LIN {X 0,Y 720.114,Z 171.461,A -85,B 0,C 180,E1 33614.463,E2 33614.463} C_VEL
